(* IEC 61131-3 sources: SmartHomeNew/ (part 8) *)

(* ---- FB_Rule_Engine.st ---- *)
FUNCTION_BLOCK FB_Rule_Engine
VAR_INPUT
    VI_System_Time_MS : UDINT;
    VI_IsActivePLC : BOOL;
    VI_Security_Armed : BOOL;
    VI_Current_Time : TOD;
    VI_Day_Of_Week : INT;
END_VAR
VAR_IN_OUT
    VI_Rules : ARRAY[1..GVL_CONSTANTS.C_MAX_RULES] OF ST_User_Rule;
    VI_Indoor_Temps : ARRAY[1..16] OF REAL;
    VI_Floor_Temps : ARRAY[1..GVL_CONSTANTS.C_MAX_HEATING_CIRCUITS] OF REAL;
    VI_Humidities : ARRAY[1..16] OF REAL;
    VI_CO2_Levels : ARRAY[1..16] OF REAL;
    VI_Motion_Sensors : ARRAY[1..16] OF BOOL;
    VI_Door_Sensors : ARRAY[1..GVL_CONSTANTS.C_MAX_DOOR_SENSORS] OF BOOL;
    VI_Window_Sensors : ARRAY[1..16] OF BOOL;
    VI_Water_Sensors : ARRAY[1..GVL_CONSTANTS.C_MAX_FLOOD_SENSORS] OF BOOL;
    VI_Smoke_Sensors : ARRAY[1..GVL_CONSTANTS.C_MAX_SMOKE_SENSORS] OF BOOL;
    VI_Methane_Sensors : ARRAY[1..GVL_CONSTANTS.C_MAX_METHANE_SENSORS] OF REAL;
    VI_CO_Sensors : ARRAY[1..GVL_CONSTANTS.C_MAX_CO_SENSORS] OF REAL;
END_VAR
VAR_OUTPUT
    VO_Preheat_Request : BOOL;
    VO_Actions : ARRAY[1..GVL_CONSTANTS.C_MAX_RULES] OF ST_Rule_Action;
END_VAR
VAR
    L_i : INT;
    L_Condition_Met : BOOL;
    L_Current_Value : REAL;
    L_Triggers : ARRAY[1..GVL_CONSTANTS.C_MAX_RULES] OF R_TRIG;
    L_Trigger_Count : ARRAY[1..GVL_CONSTANTS.C_MAX_RULES] OF UINT;
    L_Last_Reset_Time : UDINT;
    L_Elapsed_Time : UDINT;
END_VAR

IF NOT VI_IsActivePLC THEN
    FOR L_i := 1 TO GVL_CONSTANTS.C_MAX_RULES DO
        VO_Actions[L_i].Active := FALSE;
        VO_Actions[L_i].Triggered := FALSE;
        VO_Actions[L_i].Action_Type := E_Rule_Action_Type.ACTION_NONE;
        VO_Actions[L_i].Target_ID := 0;
        VO_Actions[L_i].Value := 0.0;
    END_FOR;
    VO_Preheat_Request := FALSE;
    RETURN;
END_IF;

VO_Preheat_Request := FALSE;

L_Elapsed_Time := SEL(VI_System_Time_MS >= L_Last_Reset_Time, VI_System_Time_MS - L_Last_Reset_Time, (4294967295 - L_Last_Reset_Time) + VI_System_Time_MS + 1);

IF L_Elapsed_Time >= GVL_CONSTANTS.C_MS_IN_MINUTE THEN
    L_Last_Reset_Time := VI_System_Time_MS;
    FOR L_i := 1 TO GVL_CONSTANTS.C_MAX_RULES DO
        L_Trigger_Count[L_i] := 0;
    END_FOR;
END_IF;

FOR L_i := 1 TO GVL_CONSTANTS.C_MAX_RULES DO

    // Full per-cycle action reset prevents stale Triggered/Action_Type/Target_ID/Value
    // from being observed by any downstream consumer when a rule is disabled or inactive.
    VO_Actions[L_i].Active := FALSE;
    VO_Actions[L_i].Triggered := FALSE;
    VO_Actions[L_i].Action_Type := E_Rule_Action_Type.ACTION_NONE;
    VO_Actions[L_i].Target_ID := 0;
    VO_Actions[L_i].Value := 0.0;

    IF VI_Rules[L_i].Enabled THEN
        L_Condition_Met := FALSE;
        L_Current_Value := 0.0;

        IF VI_Rules[L_i].Condition_Target_ID > 0 THEN
            CASE VI_Rules[L_i].Condition_Type OF
                E_Rule_Condition_Type.COND_AIR_TEMP:
                    IF VI_Rules[L_i].Condition_Target_ID <= 16 THEN
                        L_Current_Value := VI_Indoor_Temps[VI_Rules[L_i].Condition_Target_ID];
                    END_IF;
                E_Rule_Condition_Type.COND_FLOOR_TEMP:
                    IF VI_Rules[L_i].Condition_Target_ID <= GVL_CONSTANTS.C_MAX_HEATING_CIRCUITS THEN
                        L_Current_Value := VI_Floor_Temps[VI_Rules[L_i].Condition_Target_ID];
                    END_IF;
                E_Rule_Condition_Type.COND_HUMIDITY:
                    IF VI_Rules[L_i].Condition_Target_ID <= 16 THEN
                        L_Current_Value := VI_Humidities[VI_Rules[L_i].Condition_Target_ID];
                    END_IF;
                E_Rule_Condition_Type.COND_CO2:
                    IF VI_Rules[L_i].Condition_Target_ID <= 16 THEN
                        L_Current_Value := VI_CO2_Levels[VI_Rules[L_i].Condition_Target_ID];
                    END_IF;
                E_Rule_Condition_Type.COND_MOTION:
                    IF VI_Rules[L_i].Condition_Target_ID <= 16 THEN
                        L_Current_Value := SEL(VI_Motion_Sensors[VI_Rules[L_i].Condition_Target_ID], 0.0, 1.0);
                    END_IF;
                E_Rule_Condition_Type.COND_DOOR_WINDOW:
                    IF VI_Rules[L_i].Condition_Target_ID <= GVL_CONSTANTS.C_MAX_DOOR_SENSORS THEN
                        L_Current_Value := SEL(VI_Door_Sensors[VI_Rules[L_i].Condition_Target_ID] OR VI_Window_Sensors[VI_Rules[L_i].Condition_Target_ID], 0.0, 1.0);
                    ELSIF VI_Rules[L_i].Condition_Target_ID <= 16 THEN
                        L_Current_Value := SEL(VI_Window_Sensors[VI_Rules[L_i].Condition_Target_ID], 0.0, 1.0);
                    END_IF;
                E_Rule_Condition_Type.COND_FLOOD:
                    IF VI_Rules[L_i].Condition_Target_ID <= GVL_CONSTANTS.C_MAX_FLOOD_SENSORS THEN
                        L_Current_Value := SEL(VI_Water_Sensors[VI_Rules[L_i].Condition_Target_ID], 0.0, 1.0);
                    END_IF;
                E_Rule_Condition_Type.COND_SMOKE:
                    IF VI_Rules[L_i].Condition_Target_ID <= GVL_CONSTANTS.C_MAX_SMOKE_SENSORS THEN
                        L_Current_Value := SEL(VI_Smoke_Sensors[VI_Rules[L_i].Condition_Target_ID], 0.0, 1.0);
                    END_IF;
                E_Rule_Condition_Type.COND_METHANE:
                    IF VI_Rules[L_i].Condition_Target_ID <= GVL_CONSTANTS.C_MAX_METHANE_SENSORS THEN
                        L_Current_Value := VI_Methane_Sensors[VI_Rules[L_i].Condition_Target_ID];
                    END_IF;
                E_Rule_Condition_Type.COND_CO:
                    IF VI_Rules[L_i].Condition_Target_ID <= GVL_CONSTANTS.C_MAX_CO_SENSORS THEN
                        L_Current_Value := VI_CO_Sensors[VI_Rules[L_i].Condition_Target_ID];
                    END_IF;
                E_Rule_Condition_Type.COND_TIME_OF_DAY:
                    L_Current_Value := TO_REAL(TOD_TO_UDINT(VI_Current_Time) / GVL_CONSTANTS.C_MS_IN_MINUTE);
                E_Rule_Condition_Type.COND_DAY_OF_WEEK:
                    L_Current_Value := TO_REAL(VI_Day_Of_Week);
            END_CASE;
        ELSE
            IF VI_Rules[L_i].Condition_Type = E_Rule_Condition_Type.COND_TIME_OF_DAY THEN
                L_Current_Value := TO_REAL(TOD_TO_UDINT(VI_Current_Time) / GVL_CONSTANTS.C_MS_IN_MINUTE);
            ELSIF VI_Rules[L_i].Condition_Type = E_Rule_Condition_Type.COND_DAY_OF_WEEK THEN
                L_Current_Value := TO_REAL(VI_Day_Of_Week);
            END_IF;
        END_IF;

        CASE VI_Rules[L_i].Condition_Op OF
            E_Rule_Comparison.COMP_GT:
                L_Condition_Met := (L_Current_Value > VI_Rules[L_i].Condition_Value);
            E_Rule_Comparison.COMP_LT:
                L_Condition_Met := (L_Current_Value < VI_Rules[L_i].Condition_Value);
            E_Rule_Comparison.COMP_EQ:
                L_Condition_Met := (ABS(L_Current_Value - VI_Rules[L_i].Condition_Value) < 0.1);
            E_Rule_Comparison.COMP_GE:
                L_Condition_Met := (L_Current_Value >= VI_Rules[L_i].Condition_Value);
            E_Rule_Comparison.COMP_LE:
                L_Condition_Met := (L_Current_Value <= VI_Rules[L_i].Condition_Value);
            E_Rule_Comparison.COMP_IN_RANGE:
                L_Condition_Met := (L_Current_Value >= VI_Rules[L_i].Condition_Value) AND (L_Current_Value <= VI_Rules[L_i].Condition_Value_Max);
            E_Rule_Comparison.COMP_TRUE:
                L_Condition_Met := (L_Current_Value > 0.5);
            E_Rule_Comparison.COMP_FALSE:
                L_Condition_Met := (L_Current_Value < 0.5);
        END_CASE;

        L_Triggers[L_i](CLK := L_Condition_Met);

        IF L_Triggers[L_i].Q THEN
            L_Trigger_Count[L_i] := L_Trigger_Count[L_i] + 1;
            IF L_Trigger_Count[L_i] > 10 THEN
                CONTINUE;
            END_IF;
        END_IF;

        IF L_Condition_Met AND (L_Trigger_Count[L_i] <= 10) THEN
            VO_Actions[L_i].Active := TRUE;
            VO_Actions[L_i].Triggered := L_Triggers[L_i].Q;
            VO_Actions[L_i].Action_Type := VI_Rules[L_i].Action_Type;
            VO_Actions[L_i].Target_ID := VI_Rules[L_i].Action_Target_ID;
            VO_Actions[L_i].Value := VI_Rules[L_i].Action_Value;

            // Bridge rule-driven heating intent to policy. Per-circuit valve
            // projection remains owned by FB_Heating_Circuit_Control.
            IF (VI_Rules[L_i].Action_Type = E_Rule_Action_Type.ACTION_SET_FLOOR_HEATING) AND
               (VI_Rules[L_i].Action_Value > REAL#0.5) THEN
                VO_Preheat_Request := TRUE;
            END_IF;
        END_IF;
    END_IF;
END_FOR;

// >>> BULK_SYNC_ANCHOR: FB_Rule_Engine <<<
END_FUNCTION_BLOCK

(* ---- FB_Runtime_Bus_Replication.st ---- *)
FUNCTION_BLOCK FB_Runtime_Bus_Replication
VAR_INPUT
    VI_Enable : BOOL;
    VI_System_Time_MS : UDINT;
END_VAR
VAR
    L_Frame : ST_Runtime_Bus_Frame;
    L_TX_Index : UINT;

    L_Finalized_Runtime_Continuity : BOOL;
END_VAR

IF NOT VI_Enable THEN
    GVL_Runtime_Bus.G_Runtime_Valid := FALSE;
    RETURN;
END_IF;

// Finalized runtime continuity proof chain.
L_Finalized_Runtime_Continuity :=
    GVL_SEMANTIC_PROGRESS.Semantic_Forward_Progress_Valid
    AND GVL_SEMANTIC_PROGRESS.Semantic_Execution_Continuity_OK
    AND NOT GVL_SEMANTIC_PROGRESS.Semantic_Progress_Lease_Expired
    AND NOT GVL_SEMANTIC_PROGRESS.Semantic_Progress_Quarantine_Active
    AND GVL_RUNTIME_SNAPSHOT.Snapshot_Frozen
    AND GVL_RUNTIME_SNAPSHOT.Snapshot_Publication_Allowed
    AND GVL_RUNTIME_SNAPSHOT.Snapshot_Copy_Valid
    AND GVL_RUNTIME_SNAPSHOT.Snapshot_Isolation_Valid
    AND NOT GVL_RUNTIME_SNAPSHOT.Snapshot_Mutation_Detected
    AND GVL_DISTRIBUTED_SNAPSHOT.Distributed_Publication_Reconciled
    AND GVL_DISTRIBUTED_SNAPSHOT.Distributed_Publication_Freeze_Valid
    AND GVL_DISTRIBUTED_SNAPSHOT.Distributed_Snapshot_Consistent
    AND GVL_DISTRIBUTED_COMMIT.Distributed_Commit_Valid
    AND GVL_DISTRIBUTED_COMMIT.Publication_Prepare_Valid
    AND GVL_DISTRIBUTED_COMMIT.Publication_Commit_Confirmed
    AND NOT GVL_DISTRIBUTED_COMMIT.Peer_Commit_Mismatch
    AND NOT GVL_DISTRIBUTED_COMMIT.Commit_Lease_Expired
    AND GVL_OUTPUT_EPOCH.Output_Publication_Valid
    AND GVL_OUTPUT_EPOCH.Output_Runtime_Epoch_Valid
    AND NOT GVL_OUTPUT_EPOCH.Output_Lease_Expired
    AND NOT GVL_OUTPUT_EPOCH.Output_Forced_Safe_Decay
    AND GVL_COMMAND_VERIFY.PreOutput_Barrier_OK
    AND NOT GVL_COMMAND_VERIFY.PreOutput_Block_IO;

// Deterministic runtime replication frame publication.
L_TX_Index := GVL_Runtime_Bus.G_Last_Sequence_Id + 1;

IF L_TX_Index > 128 THEN
    L_TX_Index := 1;
END_IF;

L_Frame := (Frame_Valid := TRUE);

L_Frame.Frame_Time_MS := VI_System_Time_MS;
L_Frame.Frame_Id := GVL_Runtime_Bus.G_Last_Frame_Id + 1;

L_Frame.Source_Controller_Id :=
    GVL_Distributed_Runtime.G_Local_Node_State.Controller_Id;

L_Frame.Source_Runtime_Node_Id :=
    GVL_Distributed_Runtime.G_Local_Node_State.Runtime_Node_Id;

L_Frame.Frame_Sequence_Id :=
    GVL_Runtime_Bus.G_Last_Sequence_Id + 1;

L_Frame.Frame_Ack_Required := TRUE;

// Replicated semantic domains.
L_Frame.Authority_State_Frame := TRUE;
L_Frame.Recovery_State_Frame := TRUE;
L_Frame.Quarantine_State_Frame := TRUE;
L_Frame.Topology_State_Frame := TRUE;
L_Frame.Binding_State_Frame := TRUE;
L_Frame.Predictive_State_Frame := TRUE;

// Deterministic replication safety.
IF GVL_Distributed_Authority.G_Distributed_Safety_Barrier_OK
   AND NOT GVL_Distributed_Runtime.G_Split_Brain_Suspected
   AND L_Finalized_Runtime_Continuity THEN

    L_Frame.Replication_Consistent := TRUE;

    L_Frame.Status_Code := 0;
    L_Frame.Status_Text :=
        'Deterministic replication frame accepted';

ELSE

    L_Frame.Replication_Rejected := TRUE;

    L_Frame.Status_Code := 2;
    L_Frame.Status_Text :=
        'Deterministic replication frame rejected';

END_IF;

GVL_Runtime_Bus.G_TX_Frames[L_TX_Index] := L_Frame;

GVL_Runtime_Bus.G_Last_Frame_Id :=
    L_Frame.Frame_Id;

GVL_Runtime_Bus.G_Last_Sequence_Id :=
    L_Frame.Frame_Sequence_Id;

GVL_Runtime_Bus.G_TX_Healthy :=
    L_Frame.Replication_Consistent;

GVL_Runtime_Bus.G_RX_Healthy := TRUE;

GVL_Runtime_Bus.G_Any_Replication_Rejected :=
    L_Frame.Replication_Rejected;

GVL_Runtime_Bus.G_Runtime_Valid := TRUE;
GVL_Runtime_Bus.G_Last_Update_MS := VI_System_Time_MS;

IF L_Frame.Replication_Rejected THEN
    GVL_Runtime_Bus.G_Status_Code := 2;
    GVL_Runtime_Bus.G_Status_Text :=
        'Runtime bus replication rejected';
ELSE
    GVL_Runtime_Bus.G_Status_Code := 0;
    GVL_Runtime_Bus.G_Status_Text :=
        'Runtime bus replication healthy';
END_IF;

END_FUNCTION_BLOCK

(* ---- FB_Runtime_Node_Discovery.st ---- *)
FUNCTION_BLOCK FB_Runtime_Node_Discovery
VAR_INPUT
    VI_Enable : BOOL;
    VI_System_Time_MS : UDINT;
END_VAR
VAR
    L_i : INT;
    L_State : ST_Runtime_Node_Discovery_State;

    L_Any_Quarantine : BOOL;
    L_Any_Rejected : BOOL;
END_VAR

IF NOT VI_Enable THEN
    GVL_Runtime_Discovery.G_Runtime_Valid := FALSE;
    RETURN;
END_IF;

FOR L_i := 1 TO 32 DO

    L_State := GVL_Runtime_Discovery.G_Discovery_State[L_i];

    IF L_State.Discovery_Active THEN

        L_State.Runtime_Valid := TRUE;
        L_State.Runtime_System_Time_MS := VI_System_Time_MS;

        L_State.Node_Discovered := TRUE;

        IF GVL_Distributed_Authority.G_Distributed_Safety_Barrier_OK
           AND NOT GVL_Runtime_Sessions.G_Any_Stale_Session THEN

            L_State.Node_Validated := TRUE;
            L_State.Node_Authorized := TRUE;

            L_State.Capability_Validated := TRUE;
            L_State.Execution_Domain_Assigned := TRUE;
            L_State.Deployment_Assigned := TRUE;

            L_State.Status_Code := 0;
            L_State.Status_Text :=
                'Runtime node discovery healthy';

        ELSE

            L_State.Node_Quarantined := TRUE;
            L_State.Discovery_Rejected := TRUE;

            L_Any_Quarantine := TRUE;
            L_Any_Rejected := TRUE;

            L_State.Status_Code := 2;
            L_State.Status_Text :=
                'Runtime node discovery rejected';

        END_IF;

        GVL_Runtime_Discovery.G_Discovery_State[L_i] :=
            L_State;

    END_IF;

END_FOR;

GVL_Runtime_Discovery.G_Any_Node_Quarantined :=
    L_Any_Quarantine;

GVL_Runtime_Discovery.G_Any_Discovery_Rejected :=
    L_Any_Rejected;

GVL_Runtime_Discovery.G_Runtime_Valid := TRUE;
GVL_Runtime_Discovery.G_Last_Update_MS := VI_System_Time_MS;

IF L_Any_Rejected THEN
    GVL_Runtime_Discovery.G_Status_Code := 2;
    GVL_Runtime_Discovery.G_Status_Text :=
        'Runtime discovery rejection detected';
ELSIF L_Any_Quarantine THEN
    GVL_Runtime_Discovery.G_Status_Code := 1;
    GVL_Runtime_Discovery.G_Status_Text :=
        'Runtime discovery quarantine active';
ELSE
    GVL_Runtime_Discovery.G_Status_Code := 0;
    GVL_Runtime_Discovery.G_Status_Text :=
        'Runtime discovery governance healthy';
END_IF;

END_FUNCTION_BLOCK

(* ---- FB_Runtime_Restart_Continuity.st ---- *)
FUNCTION_BLOCK FB_Runtime_Restart_Continuity
VAR_INPUT
    VI_Enable : BOOL;
    VI_System_Time_MS : UDINT;
    VI_Warm_Restart : BOOL;
END_VAR
VAR
    L_State : ST_Runtime_Restart_Continuity_State;
END_VAR

IF NOT VI_Enable THEN
    GVL_Runtime_Restart_Continuity.G_Runtime_Valid := FALSE;
    RETURN;
END_IF;

L_State := (Runtime_Valid := TRUE);
L_State.Runtime_System_Time_MS := VI_System_Time_MS;

L_State.Warm_Restart_Detected := VI_Warm_Restart;
L_State.Cold_Start_Detected := NOT VI_Warm_Restart;

L_State.Active_Config_Version :=
    GVL_Water_Topology_Config.G_Active_Config_Version;

L_State.Restored_Config_Version :=
    GVL_Runtime_Restart_Continuity.G_Last_Stable_Config_Version;

L_State.Last_Stable_Config_Version :=
    GVL_Runtime_Restart_Continuity.G_Last_Stable_Config_Version;

L_State.Restore_Requested :=
    GVL_Runtime_Restart_Continuity.G_Restore_Request;

L_State.Post_Restart_Validation_Required :=
    GVL_Runtime_Restart_Continuity.G_Post_Restart_Validation_Request;

L_State.Retained_State_Valid := TRUE;
L_State.Topology_Restore_Valid := TRUE;
L_State.Config_Restore_Valid := TRUE;
L_State.Recovery_Restore_Valid := TRUE;
L_State.Quarantine_Restore_Valid := TRUE;

IF L_State.Restore_Requested THEN

    IF L_State.Retained_State_Valid
       AND L_State.Topology_Restore_Valid
       AND L_State.Config_Restore_Valid THEN

        L_State.Restore_Allowed := TRUE;
        L_State.Restore_Completed := TRUE;

        GVL_Config_Activation.G_Config_Quarantine_Active :=
            GVL_Runtime_Restart_Continuity.G_Last_Known_Quarantine_State;

        L_State.Status_Code := 1;
        L_State.Status_Text := 'Runtime continuity restored';

    ELSE

        L_State.Restore_Blocked := TRUE;
        L_State.Safe_Mode_Required := TRUE;
        L_State.Operator_Ack_Required := TRUE;

        L_State.Status_Code := 2;
        L_State.Status_Text := 'Runtime continuity restore blocked';

    END_IF;

ELSIF L_State.Post_Restart_Validation_Required THEN

    IF GVL_Water_Runtime_Hardening.G_Runtime_Valid
       AND GVL_Water_Output_Reconciliation.G_Runtime_Valid
       AND NOT GVL_Water_Output_Reconciliation.G_Any_Conflict_Detected THEN

        L_State.Post_Restart_Validation_OK := TRUE;

        L_State.Status_Code := 0;
        L_State.Status_Text := 'Post-restart validation healthy';

    ELSE

        L_State.Post_Restart_Validation_Failed := TRUE;
        L_State.Safe_Mode_Required := TRUE;

        L_State.Status_Code := 3;
        L_State.Status_Text := 'Post-restart validation failed';

    END_IF;

ELSE

    L_State.Status_Code := 0;
    L_State.Status_Text := 'Runtime restart continuity healthy';

END_IF;

GVL_Runtime_Restart_Continuity.G_Continuity_State := L_State;

GVL_Runtime_Restart_Continuity.G_Runtime_Valid := TRUE;
GVL_Runtime_Restart_Continuity.G_Last_Update_MS := VI_System_Time_MS;
GVL_Runtime_Restart_Continuity.G_Status_Code := L_State.Status_Code;
GVL_Runtime_Restart_Continuity.G_Status_Text := L_State.Status_Text;

END_FUNCTION_BLOCK

(* ---- FB_Runtime_Session_Governance.st ---- *)
FUNCTION_BLOCK FB_Runtime_Session_Governance
VAR_INPUT
    VI_Enable : BOOL;
    VI_System_Time_MS : UDINT;
END_VAR
VAR
    L_i : INT;
    L_Session : ST_Runtime_Node_Session;
    L_Any_Stale : BOOL;
    L_Any_Quarantine : BOOL;

    L_Finalized_Runtime_Continuity : BOOL;
END_VAR

IF NOT VI_Enable THEN
    GVL_Runtime_Sessions.G_Runtime_Valid := FALSE;
    RETURN;
END_IF;

// Finalized runtime continuity proof chain.
L_Finalized_Runtime_Continuity :=
    GVL_SEMANTIC_PROGRESS.Semantic_Forward_Progress_Valid
    AND GVL_SEMANTIC_PROGRESS.Semantic_Execution_Continuity_OK
    AND NOT GVL_SEMANTIC_PROGRESS.Semantic_Progress_Lease_Expired
    AND NOT GVL_SEMANTIC_PROGRESS.Semantic_Progress_Quarantine_Active
    AND GVL_RUNTIME_SNAPSHOT.Snapshot_Frozen
    AND GVL_RUNTIME_SNAPSHOT.Snapshot_Publication_Allowed
    AND GVL_RUNTIME_SNAPSHOT.Snapshot_Copy_Valid
    AND GVL_RUNTIME_SNAPSHOT.Snapshot_Isolation_Valid
    AND NOT GVL_RUNTIME_SNAPSHOT.Snapshot_Mutation_Detected
    AND GVL_DISTRIBUTED_SNAPSHOT.Distributed_Publication_Reconciled
    AND GVL_DISTRIBUTED_SNAPSHOT.Distributed_Publication_Freeze_Valid
    AND GVL_DISTRIBUTED_SNAPSHOT.Distributed_Snapshot_Consistent
    AND GVL_DISTRIBUTED_COMMIT.Distributed_Commit_Valid
    AND GVL_DISTRIBUTED_COMMIT.Publication_Prepare_Valid
    AND GVL_DISTRIBUTED_COMMIT.Publication_Commit_Confirmed
    AND NOT GVL_DISTRIBUTED_COMMIT.Peer_Commit_Mismatch
    AND NOT GVL_DISTRIBUTED_COMMIT.Commit_Lease_Expired
    AND GVL_OUTPUT_EPOCH.Output_Publication_Valid
    AND GVL_OUTPUT_EPOCH.Output_Runtime_Epoch_Valid
    AND NOT GVL_OUTPUT_EPOCH.Output_Lease_Expired
    AND NOT GVL_OUTPUT_EPOCH.Output_Forced_Safe_Decay
    AND GVL_COMMAND_VERIFY.PreOutput_Barrier_OK
    AND NOT GVL_COMMAND_VERIFY.PreOutput_Block_IO;

GVL_Runtime_Sessions.G_Local_Session.Session_Valid := TRUE;
GVL_Runtime_Sessions.G_Local_Session.Session_Connected := TRUE;
GVL_Runtime_Sessions.G_Local_Session.Last_Heartbeat_MS :=
    VI_System_Time_MS;

GVL_Runtime_Sessions.G_Local_Session.Transport_Healthy :=
    GVL_Runtime_Bus.G_TX_Healthy
    AND L_Finalized_Runtime_Continuity;

GVL_Runtime_Sessions.G_Local_Session.Runtime_Replication_Healthy :=
    GVL_Distributed_Runtime.G_Distributed_Replication_Healthy
    AND L_Finalized_Runtime_Continuity;

GVL_Runtime_Sessions.G_Local_Session.Authority_Granted :=
    GVL_Distributed_Authority.G_Authority_State.Authority_Master_Elected
    AND L_Finalized_Runtime_Continuity;

FOR L_i := 1 TO 16 DO

    L_Session := GVL_Runtime_Sessions.G_Remote_Sessions[L_i];

    IF L_Session.Session_Valid THEN

        IF (VI_System_Time_MS - L_Session.Last_Heartbeat_MS) > 30000 THEN

            L_Session.Session_Stale := TRUE;
            L_Session.Session_Reconnect_Required := TRUE;

            L_Any_Stale := TRUE;

        END_IF;

        IF NOT L_Finalized_Runtime_Continuity THEN

            L_Session.Session_Stale := TRUE;
            L_Session.Session_Quarantined := TRUE;

            L_Any_Stale := TRUE;
            L_Any_Quarantine := TRUE;

        END_IF;

        IF L_Session.Session_Quarantined THEN
            L_Any_Quarantine := TRUE;
        END_IF;

        GVL_Runtime_Sessions.G_Remote_Sessions[L_i] :=
            L_Session;

    END_IF;

END_FOR;

GVL_Runtime_Sessions.G_Any_Stale_Session :=
    L_Any_Stale;

GVL_Runtime_Sessions.G_Any_Quarantined_Session :=
    L_Any_Quarantine;

GVL_Runtime_Sessions.G_Runtime_Valid := TRUE;
GVL_Runtime_Sessions.G_Last_Update_MS := VI_System_Time_MS;

IF L_Any_Quarantine THEN
    GVL_Runtime_Sessions.G_Status_Code := 2;
    GVL_Runtime_Sessions.G_Status_Text :=
        'Quarantined runtime session detected';
ELSIF L_Any_Stale THEN
    GVL_Runtime_Sessions.G_Status_Code := 1;
    GVL_Runtime_Sessions.G_Status_Text :=
        'Stale runtime session detected';
ELSE
    GVL_Runtime_Sessions.G_Status_Code := 0;
    GVL_Runtime_Sessions.G_Status_Text :=
        'Runtime session governance healthy';
END_IF;

END_FUNCTION_BLOCK

(* ---- FB_Safety_Workflow_Manager.st ---- *)
FUNCTION_BLOCK FB_Safety_Workflow_Manager
VAR_INPUT
    VI_System_Time_MS : UDINT;
    VI_Water_Selective_Recover : BOOL;
    VI_Gas_Selective_Recover : BOOL;
    VI_Water_Valve_Test_Open : BOOL;
    VI_Water_Valve_Test_Close : BOOL;
    VI_Water_Valve_Test_Confirm : BOOL;
    VI_Gas_Valve_Test_Open : BOOL;
    VI_Gas_Valve_Test_Close : BOOL;
    VI_Gas_Valve_Test_Confirm : BOOL;
END_VAR
VAR_OUTPUT
    VO_Water_Selective_Recover_Edge : BOOL;
    VO_Gas_Selective_Recover_Edge : BOOL;
    VO_Water_Valve_Test_Open_Edge : BOOL;
    VO_Water_Valve_Test_Close_Edge : BOOL;
    VO_Water_Valve_Test_Confirm_Edge : BOOL;
    VO_Gas_Valve_Test_Open_Edge : BOOL;
    VO_Gas_Valve_Test_Close_Edge : BOOL;
    VO_Gas_Valve_Test_Confirm_Edge : BOOL;
    VO_Water_Test_Active : BOOL;
    VO_Gas_Test_Active : BOOL;
    VO_Water_Test_Timeout_Close_Required : BOOL;
    VO_Gas_Test_Timeout_Close_Required : BOOL;
END_VAR
VAR
    L_CMD_Water_Selective_Recover_Prev : BOOL;
    L_CMD_Gas_Selective_Recover_Prev : BOOL;
    L_CMD_Water_Valve_Test_Open_Prev : BOOL;
    L_CMD_Water_Valve_Test_Close_Prev : BOOL;
    L_CMD_Water_Valve_Test_Confirm_Prev : BOOL;
    L_CMD_Gas_Valve_Test_Open_Prev : BOOL;
    L_CMD_Gas_Valve_Test_Close_Prev : BOOL;
    L_CMD_Gas_Valve_Test_Confirm_Prev : BOOL;
    L_Water_Test_Active : BOOL;
    L_Water_Test_Start_MS : UDINT;
    L_Gas_Test_Active : BOOL;
    L_Gas_Test_Start_MS : UDINT;
END_VAR

VO_Water_Test_Timeout_Close_Required := FALSE;
VO_Gas_Test_Timeout_Close_Required := FALSE;

VO_Water_Selective_Recover_Edge := VI_Water_Selective_Recover AND NOT L_CMD_Water_Selective_Recover_Prev;
VO_Gas_Selective_Recover_Edge := VI_Gas_Selective_Recover AND NOT L_CMD_Gas_Selective_Recover_Prev;
VO_Water_Valve_Test_Open_Edge := VI_Water_Valve_Test_Open AND NOT L_CMD_Water_Valve_Test_Open_Prev;
VO_Water_Valve_Test_Close_Edge := VI_Water_Valve_Test_Close AND NOT L_CMD_Water_Valve_Test_Close_Prev;
VO_Water_Valve_Test_Confirm_Edge := VI_Water_Valve_Test_Confirm AND NOT L_CMD_Water_Valve_Test_Confirm_Prev;
VO_Gas_Valve_Test_Open_Edge := VI_Gas_Valve_Test_Open AND NOT L_CMD_Gas_Valve_Test_Open_Prev;
VO_Gas_Valve_Test_Close_Edge := VI_Gas_Valve_Test_Close AND NOT L_CMD_Gas_Valve_Test_Close_Prev;
VO_Gas_Valve_Test_Confirm_Edge := VI_Gas_Valve_Test_Confirm AND NOT L_CMD_Gas_Valve_Test_Confirm_Prev;

L_CMD_Water_Selective_Recover_Prev := VI_Water_Selective_Recover;
L_CMD_Gas_Selective_Recover_Prev := VI_Gas_Selective_Recover;
L_CMD_Water_Valve_Test_Open_Prev := VI_Water_Valve_Test_Open;
L_CMD_Water_Valve_Test_Close_Prev := VI_Water_Valve_Test_Close;
L_CMD_Water_Valve_Test_Confirm_Prev := VI_Water_Valve_Test_Confirm;
L_CMD_Gas_Valve_Test_Open_Prev := VI_Gas_Valve_Test_Open;
L_CMD_Gas_Valve_Test_Close_Prev := VI_Gas_Valve_Test_Close;
L_CMD_Gas_Valve_Test_Confirm_Prev := VI_Gas_Valve_Test_Confirm;

IF VO_Water_Valve_Test_Open_Edge THEN
    L_Water_Test_Active := TRUE;
    L_Water_Test_Start_MS := VI_System_Time_MS;
END_IF;

IF VO_Water_Valve_Test_Close_Edge OR VO_Water_Valve_Test_Confirm_Edge THEN
    L_Water_Test_Active := FALSE;
END_IF;

IF L_Water_Test_Active THEN
    IF (VI_System_Time_MS - L_Water_Test_Start_MS) >= 60000 THEN
        L_Water_Test_Active := FALSE;
        VO_Water_Test_Timeout_Close_Required := TRUE;
    END_IF;
END_IF;

IF VO_Gas_Valve_Test_Open_Edge THEN
    L_Gas_Test_Active := TRUE;
    L_Gas_Test_Start_MS := VI_System_Time_MS;
END_IF;

IF VO_Gas_Valve_Test_Close_Edge OR VO_Gas_Valve_Test_Confirm_Edge THEN
    L_Gas_Test_Active := FALSE;
END_IF;

IF L_Gas_Test_Active THEN
    IF (VI_System_Time_MS - L_Gas_Test_Start_MS) >= 60000 THEN
        L_Gas_Test_Active := FALSE;
        VO_Gas_Test_Timeout_Close_Required := TRUE;
    END_IF;
END_IF;

VO_Water_Test_Active := L_Water_Test_Active;
VO_Gas_Test_Active := L_Gas_Test_Active;
END_FUNCTION_BLOCK

(* ---- FB_Scenario_Manager.st ---- *)
FUNCTION_BLOCK FB_Scenario_Manager
VAR_INPUT
    VI_Preheat_Request : BOOL;
    VI_System_Time_MS : UDINT; // Системное время (мс)
    VI_Activate_Request : E_SCENARIO_TYPE; // Запрос на активацию сценария
    VI_IsActivePLC : BOOL; // Флаг: Данный ПЛК является ведущим
    VI_System_Mode : E_System_Operating_Mode; // Агрегированный режим работы системы
END_VAR
VAR_OUTPUT
    VO_Current_Scenario : E_SCENARIO_TYPE; // Текущий активный сценарий
    VO_Status_Msg : STRING(200); // Строковое сообщение о статусе
END_VAR

VAR
    L_Last_Scenario_Time : UDINT;
END_VAR

IF NOT VI_IsActivePLC THEN
    RETURN;
END_IF;

CASE VI_System_Mode OF
    E_System_Operating_Mode.MODE_SAFE_STOP,
    E_System_Operating_Mode.MODE_FREEZE_PROTECTION:
        IF VO_Current_Scenario <> E_SCENARIO_TYPE.SCENARIO_NONE THEN
            VO_Current_Scenario := E_SCENARIO_TYPE.SCENARIO_NONE;
            VO_Status_Msg := 'Сценарии принудительно отключены режимом безопасности';
        END_IF;
        RETURN;

    E_System_Operating_Mode.MODE_DEGRADED:
        VO_Status_Msg := 'Смена сценариев заблокирована: деградированный режим';
        RETURN;
ELSE
        // No fallback required
END_CASE;

IF VI_Activate_Request <> VO_Current_Scenario THEN
    // Проверка минимального времени работы сценария
    IF (VI_System_Time_MS - L_Last_Scenario_Time) >= 60000 OR VO_Current_Scenario = E_SCENARIO_TYPE.SCENARIO_NONE THEN
        // Логика переключения сценариев
        VO_Current_Scenario := VI_Activate_Request;
        L_Last_Scenario_Time := VI_System_Time_MS;

        CASE VO_Current_Scenario OF
        E_SCENARIO_TYPE.SCENARIO_NONE:
            VO_Status_Msg := 'Сценарии отключены';
        E_SCENARIO_TYPE.SCENARIO_AWAY:
            VO_Status_Msg := 'Активирован сценарий: Вне дома (Охрана + Энергосбережение)';
        E_SCENARIO_TYPE.SCENARIO_SLEEP:
            VO_Status_Msg := 'Активирован сценарий: Сон (Ночное освещение + Климат)';
        E_SCENARIO_TYPE.SCENARIO_PRESENCE:
            VO_Status_Msg := 'Активирован сценарий: Имитация присутствия';
        ELSE
        // No fallback required
END_CASE;
    END_IF;
END_IF;
// >>> BULK_SYNC_ANCHOR: FB_Scenario_Manager <<<

// --- PREHEAT SCENARIO INSERT ---
IF VI_Preheat_Request THEN
    // removed: direct heating write (moved to Heating Manager)
END_IF;
END_FUNCTION_BLOCK

(* ---- FB_Scenario_Transition_Guard.st ---- *)
FUNCTION_BLOCK FB_Scenario_Transition_Guard
VAR_INPUT
    VI_Current_Scenario : E_SCENARIO_TYPE;
    VI_Target_Scenario  : E_SCENARIO_TYPE;
END_VAR

VAR_OUTPUT
    VO_Transition_Allowed : BOOL;
    VO_Reason             : STRING(120);
END_VAR

VO_Transition_Allowed := TRUE;
VO_Reason := 'OK';

// no-op transition is always allowed
IF VI_Current_Scenario = VI_Target_Scenario THEN
    RETURN;
END_IF;

// emergency can always be entered
IF VI_Target_Scenario = E_SCENARIO_TYPE.SCENARIO_EMERGENCY THEN
    RETURN;
END_IF;

// from NONE, any target is allowed
IF VI_Current_Scenario = E_SCENARIO_TYPE.SCENARIO_NONE THEN
    RETURN;
END_IF;

// emergency exit is restricted
IF VI_Current_Scenario = E_SCENARIO_TYPE.SCENARIO_EMERGENCY THEN
    CASE VI_Target_Scenario OF
        E_SCENARIO_TYPE.SCENARIO_NONE,
        E_SCENARIO_TYPE.SCENARIO_AWAY,
        E_SCENARIO_TYPE.SCENARIO_SLEEP,
        E_SCENARIO_TYPE.SCENARIO_PRESENCE:
            RETURN;
    ELSE
        VO_Transition_Allowed := FALSE;
        VO_Reason := 'Переход из EMERGENCY в данный сценарий запрещён';
        RETURN;
    END_CASE;
END_IF;

// away exit is restricted to safe occupancy contexts
IF VI_Current_Scenario = E_SCENARIO_TYPE.SCENARIO_AWAY THEN
    CASE VI_Target_Scenario OF
        E_SCENARIO_TYPE.SCENARIO_NONE,
        E_SCENARIO_TYPE.SCENARIO_SLEEP,
        E_SCENARIO_TYPE.SCENARIO_PRESENCE,
        E_SCENARIO_TYPE.SCENARIO_EMERGENCY:
            RETURN;
    ELSE
        VO_Transition_Allowed := FALSE;
        VO_Reason := 'Переход из AWAY в данный сценарий запрещён';
        RETURN;
    END_CASE;
END_IF;

// default: allow
RETURN;
// >>> BULK_SYNC_ANCHOR: FB_Scenario_Transition_Guard <<<

(* ---- FB_Security_System_Manager.st ---- *)
FUNCTION_BLOCK FB_Security_System_Manager
VAR_INPUT
    VI_System_Time_MS : UDINT; // Системное время (мс)
    VI_IsActivePLC : BOOL; // Флаг: Данный ПЛК является ведущим
    VI_Arm_Request : BOOL; // Запрос на постановку под охрану
    VI_Disarm_Request : BOOL; // Запрос на снятие с охраны
    VI_PIN_Code : STRING(4); // ПИН-код для авторизации
    VI_RFID_Tag : STRING(20); // RFID/NFC метка для авторизации
    VI_2FA_Code : STRING(6); // Код двухфакторной аутентификации
    VI_Config : ST_Security_Global_Config; // Конфигурация охранной системы
    VI_Current_TOD : TOD; // Текущее время суток (от FB_Astro_Timer)
END_VAR
VAR_IN_OUT
    VI_Motion_Sensors : ARRAY[1..16] OF BOOL; // Датчики движения
    VI_Door_Sensors : ARRAY[1..GVL_CONSTANTS.C_MAX_DOOR_SENSORS] OF BOOL; // Датчики открытия дверей (герконы)
    VI_Window_Sensors : ARRAY[1..16] OF BOOL; // Датчики открытия окон (герконы)
    VI_Bypass_Motion : ARRAY[1..16] OF BOOL; // Байпас датчиков движения
    VI_Bypass_Doors : ARRAY[1..GVL_CONSTANTS.C_MAX_DOOR_SENSORS] OF BOOL; // Байпас дверей
    VI_Bypass_Windows : ARRAY[1..16] OF BOOL; // Байпас окон
END_VAR
VAR_OUTPUT
    VO_Armed : BOOL; // Статус: Система под охраной
    VO_Alarm_Active : BOOL; // Статус: Тревога активна
    VO_Siren_Active : BOOL; // Команда: Включить сирену
    VO_Status_Msg : STRING(200); // Строковое сообщение о статусе
    VO_Send_Code_Req : BOOL; // Запрос на отправку кода 2FA
    VO_Code_To_Send : STRING(6); // Сгенерированный код 2FA для отправки
END_VAR
VAR
    L_i : INT;
    L_Any_Sensor_Active : BOOL;
    L_Door_Blocking_Open : BOOL;
    L_Window_Blocking_Open : BOOL;
    L_Intrusion_Active_Count : INT;
    L_Intrusion_Event_Count : INT;
    L_Arm_Delay_Timer : FB_System_Timer;
    L_Alarm_Delay_Timer : FB_System_Timer;
    L_Arming_In_Progress : BOOL;
    L_Pin_Entry_Active : BOOL;
    L_Valid_PIN : BOOL;
    fbAccessCode : FB_AccessCode_Manager;
    fbTwoFactor : FB_TwoFactor_Auth;
    L_2FA_Required : BOOL;
    L_Disarm_Pending : BOOL;
    L_Reset_2FA : BOOL;
    L_Auto_Arm_Trigger : BOOL;
    L_Max_Attempts : BYTE;
    L_PIN_Fail_Count : BYTE;
    L_Pin_Entry_Timeout_MS : UDINT;
    L_Combined_Window_MS : UDINT;
    L_Combined_Elapsed_MS : UDINT;
    L_Combined_Window_Active : BOOL;
    L_Combined_First_Event_MS : UDINT;
    L_Combined_Event_Count : INT;
    L_Allowed_Open_Windows : ARRAY[1..16] OF BOOL;
    L_Prev_Motion_Sensors : ARRAY[1..16] OF BOOL;
    L_Prev_Door_Sensors : ARRAY[1..GVL_CONSTANTS.C_MAX_DOOR_SENSORS] OF BOOL;
    L_Prev_Window_Sensors : ARRAY[1..16] OF BOOL;
    R_Trig_Auto_Arm : R_TRIG;
    R_Trig_Arm : R_TRIG;
    R_Trig_Disarm : R_TRIG;
END_VAR

IF NOT VI_IsActivePLC THEN
    VO_Armed := FALSE;
    VO_Alarm_Active := FALSE;
    VO_Siren_Active := FALSE;
    VO_Send_Code_Req := FALSE;
    VO_Code_To_Send := '';
    VO_Status_Msg := 'Охрана: резервный ПЛК';
    L_Arming_In_Progress := FALSE;
    L_Disarm_Pending := FALSE;
    L_2FA_Required := FALSE;
    L_Reset_2FA := FALSE;
    L_Pin_Entry_Active := FALSE;
    GVL_SECURITY_WORKFLOW.G_Arming_In_Progress := FALSE;
    GVL_SECURITY_WORKFLOW.G_Pin_Entry_Active := FALSE;
    GVL_SECURITY_WORKFLOW.G_Disarm_Pending := FALSE;
    GVL_SECURITY_WORKFLOW.G_2FA_Required := FALSE;
    GVL_SECURITY_WORKFLOW.G_2FA_Send_Code_Req := FALSE;
    GVL_SECURITY_WORKFLOW.G_Combined_Window_Active := FALSE;
    GVL_SECURITY_WORKFLOW.G_Combined_Event_Count := 0;
    GVL_SECURITY_WORKFLOW.G_Intrusion_Active_Count := 0;
    GVL_SECURITY_WORKFLOW.G_Intrusion_Event_Count := 0;
    GVL_SECURITY_WORKFLOW.G_Any_Sensor_Active := FALSE;
    GVL_SECURITY_WORKFLOW.G_Status_Text := VO_Status_Msg;
    GVL_SECURITY_WORKFLOW.G_Last_Update_MS := VI_System_Time_MS;
    RETURN;
END_IF;

IF VI_Config.max_access_attempts < 1 THEN
    L_Max_Attempts := 1;
ELSE
    L_Max_Attempts := VI_Config.max_access_attempts;
END_IF;

IF VI_Config.pin_entry_timeout_seconds > 0 THEN
    L_Pin_Entry_Timeout_MS := VI_Config.pin_entry_timeout_seconds * 1000;
ELSIF VI_Config.entry_delay_seconds > 0 THEN
    L_Pin_Entry_Timeout_MS := VI_Config.entry_delay_seconds * 1000;
ELSE
    L_Pin_Entry_Timeout_MS := 45000;
END_IF;

IF VI_Config.combined_alarm_window_seconds > 0 THEN
    L_Combined_Window_MS := VI_Config.combined_alarm_window_seconds * 1000;
ELSE
    L_Combined_Window_MS := 10000;
END_IF;

R_Trig_Arm(CLK := VI_Arm_Request);
R_Trig_Disarm(CLK := VI_Disarm_Request);

// 1. Проверка PIN-кода или RFID-метки через менеджер кодов
fbAccessCode(
    VI_System_Time_MS := VI_System_Time_MS,
    VI_IsActivePLC := VI_IsActivePLC,
    VI_Code_To_Check := VI_PIN_Code,
    VI_RFID_To_Check := VI_RFID_Tag,
    VI_Access_Codes := GVL_RETAIN.G_Access_Codes,
    VI_RFID_Tags := GVL_RETAIN.G_RFID_Tags,
    VO_Code_Valid => L_Valid_PIN
);

// 2. Логика постановки на охрану (с задержкой на выход)
L_Auto_Arm_Trigger := FALSE;
IF VI_Config.auto_arm_enabled THEN
    IF VI_Current_TOD >= UDINT_TO_TOD(VI_Config.auto_arm_time_ms) THEN
        L_Auto_Arm_Trigger := TRUE;
    END_IF;
END_IF;
R_Trig_Auto_Arm(CLK := L_Auto_Arm_Trigger);

IF ((R_Trig_Arm.Q AND L_Valid_PIN) OR R_Trig_Auto_Arm.Q) AND NOT VO_Armed AND NOT L_Arming_In_Progress THEN
    L_Door_Blocking_Open := FALSE;
    L_Window_Blocking_Open := FALSE;

    FOR L_i := 1 TO GVL_CONSTANTS.C_MAX_DOOR_SENSORS DO
        IF VI_Door_Sensors[L_i] AND NOT VI_Bypass_Doors[L_i] THEN
            L_Door_Blocking_Open := TRUE;
        END_IF;
    END_FOR;

    FOR L_i := 1 TO 16 DO
        IF VI_Window_Sensors[L_i] AND NOT VI_Bypass_Windows[L_i] THEN
            L_Window_Blocking_Open := TRUE;
        END_IF;
    END_FOR;

    IF NOT L_Door_Blocking_Open AND (NOT L_Window_Blocking_Open OR VI_Config.allow_short_away_open_windows) THEN
        FOR L_i := 1 TO 16 DO
            L_Allowed_Open_Windows[L_i] :=
                VI_Config.allow_short_away_open_windows
                AND VI_Window_Sensors[L_i]
                AND NOT VI_Bypass_Windows[L_i];
        END_FOR;

        L_Arming_In_Progress := TRUE;
        L_PIN_Fail_Count := 0;
        L_Pin_Entry_Active := FALSE;
        L_Combined_Window_Active := FALSE;
        L_Combined_Event_Count := 0;
        VO_Status_Msg := 'Постановка на охрану. Покиньте помещение.';
    ELSE
        IF L_Door_Blocking_Open THEN
            VO_Status_Msg := 'Ошибка постановки: Открыты двери';
        ELSE
            VO_Status_Msg := 'Ошибка постановки: Открыты окна';
        END_IF;
    END_IF;
END_IF;

L_Arm_Delay_Timer(IN := L_Arming_In_Progress, PT := TO_TIME(VI_Config.exit_delay_seconds * 1000), VI_System_Time_MS := VI_System_Time_MS);
IF L_Arm_Delay_Timer.Q THEN
    L_Arming_In_Progress := FALSE;
    VO_Armed := TRUE;
    VO_Status_Msg := 'Система под охраной';
END_IF;

// 3. Логика снятия с охраны с PIN/RFID и 2FA
IF R_Trig_Disarm.Q AND VO_Armed THEN
    IF L_Valid_PIN THEN
        L_PIN_Fail_Count := 0;

        IF VI_Config.enable_2fa THEN
            L_Disarm_Pending := TRUE;
            L_2FA_Required := TRUE;
            VO_Status_Msg := 'Ожидание 2FA для снятия с охраны';
        ELSE
            VO_Armed := FALSE;
            VO_Alarm_Active := FALSE;
            VO_Siren_Active := FALSE;
            L_Arming_In_Progress := FALSE;
            L_Pin_Entry_Active := FALSE;
            L_Combined_Window_Active := FALSE;
            L_Combined_Event_Count := 0;
            FOR L_i := 1 TO 16 DO
                L_Allowed_Open_Windows[L_i] := FALSE;
            END_FOR;
            VO_Status_Msg := 'Система снята с охраны';
        END_IF;
    ELSE
        IF L_PIN_Fail_Count < 255 THEN
            L_PIN_Fail_Count := L_PIN_Fail_Count + 1;
        END_IF;

        IF L_PIN_Fail_Count >= L_Max_Attempts THEN
            VO_Alarm_Active := TRUE;
            VO_Siren_Active := TRUE;
            VO_Status_Msg := 'ТРЕВОГА! Превышено количество попыток PIN';
        ELSE
            VO_Status_Msg := 'Неверный PIN/RFID';
        END_IF;
    END_IF;
END_IF;

fbTwoFactor(
    VI_System_Time_MS := VI_System_Time_MS,
    VI_Start_Auth := L_2FA_Required,
    VI_Method := E_TwoFactor_Method.TF_METHOD_TOTP,
    VI_User_Code := VI_2FA_Code,
    VI_Reset_Success := L_Reset_2FA
);

VO_Send_Code_Req := fbTwoFactor.VO_Send_Code_Req;
VO_Code_To_Send := fbTwoFactor.VO_Code_To_Send;

IF L_Disarm_Pending AND fbTwoFactor.VO_State.Is_Success THEN
    VO_Armed := FALSE;
    VO_Alarm_Active := FALSE;
    VO_Siren_Active := FALSE;
    L_Arming_In_Progress := FALSE;
    L_Pin_Entry_Active := FALSE;
    L_Disarm_Pending := FALSE;
    L_2FA_Required := FALSE;
    L_Reset_2FA := TRUE;
    L_Combined_Window_Active := FALSE;
    L_Combined_Event_Count := 0;
    FOR L_i := 1 TO 16 DO
        L_Allowed_Open_Windows[L_i] := FALSE;
    END_FOR;
    VO_Status_Msg := 'Система снята с охраны';
ELSIF L_Disarm_Pending AND fbTwoFactor.VO_State.Is_Locked THEN
    L_Disarm_Pending := FALSE;
    L_2FA_Required := FALSE;
    L_Reset_2FA := FALSE;
    VO_Status_Msg := 'Ошибка 2FA: Превышено количество попыток';
ELSE
    L_Reset_2FA := FALSE;
END_IF;

// 4. Логика тревоги: задержка PIN + комбинированная авария датчиков
IF VO_Armed THEN
    FOR L_i := 1 TO 16 DO
        IF L_Allowed_Open_Windows[L_i] AND NOT VI_Window_Sensors[L_i] THEN
            L_Allowed_Open_Windows[L_i] := FALSE;
        END_IF;
    END_FOR;

    L_Any_Sensor_Active := FALSE;
    L_Intrusion_Active_Count := 0;
    L_Intrusion_Event_Count := 0;

    FOR L_i := 1 TO 16 DO
        IF VI_Motion_Sensors[L_i] AND NOT VI_Bypass_Motion[L_i] THEN
            L_Any_Sensor_Active := TRUE;
            L_Intrusion_Active_Count := L_Intrusion_Active_Count + 1;
            IF NOT L_Prev_Motion_Sensors[L_i] THEN
                L_Intrusion_Event_Count := L_Intrusion_Event_Count + 1;
            END_IF;
        END_IF;
        L_Prev_Motion_Sensors[L_i] := VI_Motion_Sensors[L_i];
    END_FOR;

    FOR L_i := 1 TO GVL_CONSTANTS.C_MAX_DOOR_SENSORS DO
        IF VI_Door_Sensors[L_i] AND NOT VI_Bypass_Doors[L_i] THEN
            L_Any_Sensor_Active := TRUE;
            L_Intrusion_Active_Count := L_Intrusion_Active_Count + 1;
            IF NOT L_Prev_Door_Sensors[L_i] THEN
                L_Intrusion_Event_Count := L_Intrusion_Event_Count + 1;
            END_IF;
        END_IF;
        L_Prev_Door_Sensors[L_i] := VI_Door_Sensors[L_i];
    END_FOR;

    FOR L_i := 1 TO 16 DO
        IF VI_Window_Sensors[L_i] AND NOT VI_Bypass_Windows[L_i] AND NOT L_Allowed_Open_Windows[L_i] THEN
            L_Any_Sensor_Active := TRUE;
            L_Intrusion_Active_Count := L_Intrusion_Active_Count + 1;
            IF NOT L_Prev_Window_Sensors[L_i] THEN
                L_Intrusion_Event_Count := L_Intrusion_Event_Count + 1;
            END_IF;
        END_IF;
        L_Prev_Window_Sensors[L_i] := VI_Window_Sensors[L_i];
    END_FOR;

    IF L_Intrusion_Event_Count > 0 THEN
        IF NOT L_Combined_Window_Active THEN
            L_Combined_Window_Active := TRUE;
            L_Combined_First_Event_MS := VI_System_Time_MS;
            L_Combined_Event_Count := L_Intrusion_Event_Count;
        ELSE
            IF VI_System_Time_MS >= L_Combined_First_Event_MS THEN
                L_Combined_Elapsed_MS := VI_System_Time_MS - L_Combined_First_Event_MS;
            ELSE
                L_Combined_Elapsed_MS := (4294967295 - L_Combined_First_Event_MS) + VI_System_Time_MS + 1;
            END_IF;

            IF L_Combined_Elapsed_MS <= L_Combined_Window_MS THEN
                L_Combined_Event_Count := L_Combined_Event_Count + L_Intrusion_Event_Count;
            ELSE
                L_Combined_First_Event_MS := VI_System_Time_MS;
                L_Combined_Event_Count := L_Intrusion_Event_Count;
            END_IF;
        END_IF;
    END_IF;

    IF L_Combined_Window_Active THEN
        IF VI_System_Time_MS >= L_Combined_First_Event_MS THEN
            L_Combined_Elapsed_MS := VI_System_Time_MS - L_Combined_First_Event_MS;
        ELSE
            L_Combined_Elapsed_MS := (4294967295 - L_Combined_First_Event_MS) + VI_System_Time_MS + 1;
        END_IF;

        IF L_Combined_Elapsed_MS > L_Combined_Window_MS THEN
            L_Combined_Window_Active := FALSE;
            L_Combined_Event_Count := 0;
        END_IF;
    END_IF;

    IF (L_Intrusion_Active_Count >= 2) OR (L_Combined_Window_Active AND (L_Combined_Event_Count >= 2)) THEN
        VO_Alarm_Active := TRUE;
        VO_Siren_Active := TRUE;
        L_Pin_Entry_Active := FALSE;
        VO_Status_Msg := 'ТРЕВОГА! Комбинированное нарушение периметра';
    ELSIF L_Any_Sensor_Active THEN
        L_Pin_Entry_Active := TRUE;
    END_IF;

    L_Alarm_Delay_Timer(IN := L_Pin_Entry_Active, PT := TO_TIME(L_Pin_Entry_Timeout_MS), VI_System_Time_MS := VI_System_Time_MS);

    IF L_Alarm_Delay_Timer.Q THEN
        VO_Alarm_Active := TRUE;
        VO_Siren_Active := TRUE;
        VO_Status_Msg := 'ТРЕВОГА! Нарушение периметра';
    ELSIF L_Pin_Entry_Active AND NOT VO_Alarm_Active THEN
        VO_Status_Msg := 'Внимание! Введите PIN-код для отмены тревоги';
    END_IF;
ELSE
    L_Any_Sensor_Active := FALSE;
    L_Intrusion_Active_Count := 0;
    L_Intrusion_Event_Count := 0;
    L_Pin_Entry_Active := FALSE;
    L_Alarm_Delay_Timer(IN := FALSE, PT := T#0s, VI_System_Time_MS := VI_System_Time_MS);
END_IF;

GVL_SECURITY_WORKFLOW.G_Arming_In_Progress := L_Arming_In_Progress;
GVL_SECURITY_WORKFLOW.G_Arm_Delay_ET := L_Arm_Delay_Timer.ET;
GVL_SECURITY_WORKFLOW.G_Arm_Delay_Q := L_Arm_Delay_Timer.Q;
GVL_SECURITY_WORKFLOW.G_Pin_Entry_Active := L_Pin_Entry_Active;
GVL_SECURITY_WORKFLOW.G_Entry_Delay_ET := L_Alarm_Delay_Timer.ET;
GVL_SECURITY_WORKFLOW.G_Entry_Delay_Q := L_Alarm_Delay_Timer.Q;
GVL_SECURITY_WORKFLOW.G_Pin_Fail_Count := L_PIN_Fail_Count;
GVL_SECURITY_WORKFLOW.G_Max_Attempts := L_Max_Attempts;
GVL_SECURITY_WORKFLOW.G_Disarm_Pending := L_Disarm_Pending;
GVL_SECURITY_WORKFLOW.G_2FA_Required := L_2FA_Required;
GVL_SECURITY_WORKFLOW.G_2FA_Send_Code_Req := VO_Send_Code_Req;
GVL_SECURITY_WORKFLOW.G_Combined_Window_Active := L_Combined_Window_Active;
GVL_SECURITY_WORKFLOW.G_Combined_Event_Count := L_Combined_Event_Count;
GVL_SECURITY_WORKFLOW.G_Intrusion_Active_Count := L_Intrusion_Active_Count;
GVL_SECURITY_WORKFLOW.G_Intrusion_Event_Count := L_Intrusion_Event_Count;
GVL_SECURITY_WORKFLOW.G_Any_Sensor_Active := L_Any_Sensor_Active;
GVL_SECURITY_WORKFLOW.G_Door_Blocking_Open := L_Door_Blocking_Open;
GVL_SECURITY_WORKFLOW.G_Window_Blocking_Open := L_Window_Blocking_Open;
GVL_SECURITY_WORKFLOW.G_Status_Text := VO_Status_Msg;
GVL_SECURITY_WORKFLOW.G_Last_Update_MS := VI_System_Time_MS;

// >>> BULK_SYNC_ANCHOR: FB_Security_System_Manager <<<
END_FUNCTION_BLOCK

(* ---- FB_Sensor_Calibration.st ---- *)
FUNCTION_BLOCK FB_Sensor_Calibration
VAR_INPUT
    VI_Sensor_ID : UDINT;
    VI_Reference_Value : REAL;
    VI_Current_Value : REAL;
    VI_Apply : BOOL;
END_VAR
VAR_OUTPUT
    VO_Offset : REAL;
    VO_Multiplier : REAL := 1.0;
    VO_Done : BOOL;
END_VAR
VAR
    L_Applied : BOOL;
END_VAR

IF VI_Apply AND NOT L_Applied THEN
    // Простая калибровка смещением (одноточечная)
    VO_Offset := VI_Reference_Value - VI_Current_Value;
    VO_Done := TRUE;
    L_Applied := TRUE;
ELSIF NOT VI_Apply THEN
    VO_Done := FALSE;
    L_Applied := FALSE;
END_IF;
END_FUNCTION_BLOCK

(* ---- FB_Sensor_Calibration_Processor.st ---- *)
FUNCTION_BLOCK FB_Sensor_Calibration_Processor
VAR_INPUT
    VI_Raw_Value : REAL;
    VI_Record    : ST_Sensor_Calibration_Record;
END_VAR
VAR_OUTPUT
    VO_Calibrated_Value : REAL;
END_VAR

VO_Calibrated_Value := (VI_Raw_Value * VI_Record.multiplier) + VI_Record.offset;

(* ---- FB_Simulation_Manager.st ---- *)
FUNCTION_BLOCK FB_Simulation_Manager
VAR_INPUT
    VI_System_Time_MS : UDINT; // Системное время (мс)
    VI_IsActivePLC    : BOOL; // Флаг: Данный ПЛК является ведущим
    VI_Scenario       : E_SCENARIO_TYPE; // Текущий активный сценарий
    VI_Config         : ST_Scenario_Config; // Конфигурация сценариев
END_VAR
VAR_OUTPUT
    VO_Sim_Lights     : ARRAY[1..32] OF BOOL; // Симулированные сигналы включения света
    VO_Sim_Active     : BOOL; // Флаг: Симуляция присутствия активна
    // Симуляция аварий (для тестирования)
    VO_Sim_Water_Leak : ARRAY[1..GVL_CONSTANTS.C_MAX_FLOOD_SENSORS] OF BOOL; // Симулированные сигналы протечки
    VO_Sim_Gas_Leak   : ARRAY[1..GVL_CONSTANTS.C_MAX_METHANE_SENSORS] OF REAL; // Симулированные уровни газа
END_VAR
VAR
    L_Random          : FB_Random_Generator;
    L_Last_Toggle     : UDINT;
    L_i               : INT;
    L_Rand_Val        : UDINT;
    L_Test_Mode       : BOOL := FALSE; // Флаг тестового режима
END_VAR

IF VI_Scenario = E_SCENARIO_TYPE.SCENARIO_AWAY AND VI_Config.Presence_Simulation_Enabled THEN
    VO_Sim_Active := TRUE;

    // Переключаем свет каждые 30 минут
    IF (VI_System_Time_MS - L_Last_Toggle) >= (GVL_CONSTANTS.C_MS_IN_MINUTE * 30) THEN
        L_Last_Toggle := VI_System_Time_MS;

        FOR L_i := 1 TO 32 DO
            L_Rand_Val := 1;
            VO_Sim_Lights[L_i] := (L_Rand_Val > 80); // 20% шанс включения
        END_FOR;
    END_IF;
ELSE
    VO_Sim_Active := FALSE;
    FOR L_i := 1 TO 32 DO VO_Sim_Lights[L_i] := FALSE; END_FOR;
END_IF;

// Симуляция аварий в тестовом режиме
IF L_Test_Mode THEN
    // Генерация случайных протечек (очень редко)
    L_Rand_Val := 1;
    IF L_Rand_Val = 42 THEN
        VO_Sim_Water_Leak[1] := TRUE;
    END_IF;

    // Симуляция утечки газа
    L_Rand_Val := 1;
    IF L_Rand_Val = 77 THEN
        VO_Sim_Gas_Leak[1] := 15.0; // 15% LEL
    END_IF;
ELSE
    FOR L_i := 1 TO GVL_CONSTANTS.C_MAX_FLOOD_SENSORS DO VO_Sim_Water_Leak[L_i] := FALSE; END_FOR;
    FOR L_i := 1 TO GVL_CONSTANTS.C_MAX_METHANE_SENSORS DO VO_Sim_Gas_Leak[L_i] := 0.0; END_FOR;
END_IF;
// >>> BULK_SYNC_ANCHOR: FB_Simulation_Manager <<<

(* ---- FB_Smoke_Detector.st ---- *)
FUNCTION_BLOCK FB_Smoke_Detector
VAR_INPUT
    VI_Smoke_Signal : BOOL;
END_VAR
VAR_OUTPUT
    VO_Smoke_Detected : BOOL;
END_VAR

VO_Smoke_Detected := VI_Smoke_Signal;

(* ---- FB_Socket_Manager.st ---- *)
FUNCTION_BLOCK FB_Socket_Manager
VAR_INPUT
    VI_System_Time_MS : UDINT;
    VI_IsActivePLC : BOOL;
    VI_Scenario : E_SCENARIO_TYPE;
    VI_Fire_Alarm : BOOL;
    VI_Flood_Alarm : BOOL;
    VI_Security_Armed : BOOL;
END_VAR
VAR_IN_OUT
    VI_Manual_Override : ARRAY[1..GVL_CONSTANTS.C_MAX_SOCKETS] OF BOOL;
    VI_Physical_Switches : ARRAY[1..GVL_CONSTANTS.C_MAX_SOCKETS] OF BOOL;
    VI_Rule_Actions : ARRAY[1..GVL_CONSTANTS.C_MAX_RULES] OF ST_Rule_Action;
    VI_IO_Modules_Online : ARRAY[1..GVL_CONSTANTS.C_MAX_MODULES] OF BOOL;
END_VAR
VAR_OUTPUT
    VO_Socket_States : ARRAY[1..GVL_CONSTANTS.C_MAX_SOCKETS] OF BOOL;
    VO_Internal_States : ARRAY[1..GVL_CONSTANTS.C_MAX_SOCKETS] OF BOOL;
END_VAR
VAR
    L_i : INT;
    L_j : INT;
    L_Rule_State : BOOL;
    L_Rule_Active : BOOL;
    L_Internal_State : ARRAY[1..GVL_CONSTANTS.C_MAX_SOCKETS] OF BOOL;
    L_Manual_Trig : ARRAY[1..GVL_CONSTANTS.C_MAX_SOCKETS] OF R_TRIG;
END_VAR

FOR L_i := 1 TO GVL_CONSTANTS.C_MAX_SOCKETS DO
    VO_Socket_States[L_i] := FALSE;
    VO_Internal_States[L_i] := L_Internal_State[L_i];
END_FOR;

IF NOT VI_IsActivePLC THEN
    RETURN;
END_IF;

FOR L_i := 1 TO GVL_CONSTANTS.C_MAX_MODULES DO
    IF NOT VI_IO_Modules_Online[L_i] THEN
        RETURN;
    END_IF;
END_FOR;

FOR L_i := 1 TO GVL_CONSTANTS.C_MAX_SOCKETS DO
    L_Rule_Active := FALSE;
    L_Rule_State := FALSE;

    L_Manual_Trig[L_i](CLK := VI_Manual_Override[L_i]);

    IF L_Manual_Trig[L_i].Q THEN
        L_Internal_State[L_i] := NOT L_Internal_State[L_i];
    END_IF;

    FOR L_j := 1 TO GVL_CONSTANTS.C_MAX_RULES DO
        IF VI_Rule_Actions[L_j].Active AND VI_Rule_Actions[L_j].Target_ID = L_i THEN
            IF VI_Rule_Actions[L_j].Action_Type = E_Rule_Action_Type.ACTION_SET_SOCKET THEN
                L_Rule_Active := TRUE;
                L_Rule_State := (VI_Rule_Actions[L_j].Value > 0.5);
                L_Internal_State[L_i] := L_Rule_State;
            ELSIF VI_Rule_Actions[L_j].Action_Type = E_Rule_Action_Type.ACTION_TOGGLE_SOCKET AND VI_Rule_Actions[L_j].Triggered THEN
                L_Internal_State[L_i] := NOT L_Internal_State[L_i];
            END_IF;
        END_IF;
    END_FOR;

    IF VI_Fire_Alarm OR VI_Flood_Alarm THEN
        IF L_i > 4 THEN
            VO_Socket_States[L_i] := FALSE;
        ELSE
            VO_Socket_States[L_i] := L_Internal_State[L_i];
        END_IF;
    ELSIF VI_Scenario = E_SCENARIO_TYPE.SCENARIO_AWAY OR VI_Security_Armed THEN
        IF L_i > 4 THEN
            VO_Socket_States[L_i] := FALSE;
        ELSE
            VO_Socket_States[L_i] := L_Internal_State[L_i];
        END_IF;
    ELSE
        IF L_Rule_Active THEN
            VO_Socket_States[L_i] := L_Rule_State;
        ELSE
            VO_Socket_States[L_i] := L_Internal_State[L_i];
        END_IF;
    END_IF;
END_FOR;

VO_Internal_States := L_Internal_State;

END_FUNCTION_BLOCK
// >>> BULK_SYNC_ANCHOR: FB_Socket_Manager <<<

(* ---- FB_Socket_V2_Staging.st ---- *)
FUNCTION_BLOCK FB_Socket_V2_Staging
VAR_INPUT
    VI_Socket_ID : INT;
    VI_Enable : BOOL;
    VI_Target_State : BOOL;
    VI_Manual_Override : BOOL;
    VI_Safety_Lock : BOOL;
    VI_Scenario_ID : INT;
    VI_Is_On : BOOL;
    VI_Manual_Override_Active : BOOL;
    VI_Safety_Blocked : BOOL;
    VI_Alarm_Active : BOOL;
END_VAR
VAR_OUTPUT
    VO_Command_Shadow : ST_Socket_Command_V2;
    VO_State_Shadow : ST_Socket_State_V2;
END_VAR

VO_Command_Shadow.Target_State := VI_Target_State;
VO_State_Shadow.Is_On := VI_Is_On;
VO_State_Shadow.Safety_Blocked := VI_Safety_Blocked;
END_FUNCTION_BLOCK

(* ---- FB_State_Manager.st ---- *)
FUNCTION_BLOCK FB_State_Manager
VAR_INPUT
    VI_System_Severity : E_System_Severity;
    VI_Root_Cause      : E_System_Root_Cause;
    VI_Freeze_Risk     : BOOL := FALSE;
END_VAR

VAR_OUTPUT
    VO_System_OK        : BOOL;
    VO_System_Warning   : BOOL;
    VO_System_Critical  : BOOL;
    VO_Status_Msg       : STRING(200);

    // compatibility output for existing orchestration
    VO_System_Mode      : E_System_Operating_Mode;
END_VAR

VO_System_OK := FALSE;
VO_System_Warning := FALSE;
VO_System_Critical := FALSE;
VO_Status_Msg := '';
VO_System_Mode := E_System_Operating_Mode.MODE_NORMAL;

CASE VI_System_Severity OF
    E_System_Severity.SEV_NORMAL:
        VO_System_OK := TRUE;
        VO_Status_Msg := 'Система в норме';
        VO_System_Mode := E_System_Operating_Mode.MODE_NORMAL;

    E_System_Severity.SEV_WARNING:
        VO_System_Warning := TRUE;
        VO_System_Mode := E_System_Operating_Mode.MODE_DEGRADED;
        CASE VI_Root_Cause OF
            E_System_Root_Cause.ROOT_WATER_LEAK:
                VO_Status_Msg := 'Предупреждение: протечка воды';
            E_System_Root_Cause.ROOT_CO_WARNING:
                VO_Status_Msg := 'Предупреждение: повышенный CO';
            ELSE
                VO_Status_Msg := 'Предупреждение системы';
        END_CASE;

    E_System_Severity.SEV_DEGRADED:
        VO_System_Warning := TRUE;
        VO_System_Mode := E_System_Operating_Mode.MODE_DEGRADED;
        CASE VI_Root_Cause OF
            E_System_Root_Cause.ROOT_SENSOR_FAULT:
                VO_Status_Msg := 'Деградация: ошибка датчика';
            E_System_Root_Cause.ROOT_IO_OFFLINE:
                VO_Status_Msg := 'Деградация: модуль IO недоступен';
            E_System_Root_Cause.ROOT_COMM_FAULT:
                VO_Status_Msg := 'Деградация: ошибка связи';
            E_System_Root_Cause.ROOT_WATCHDOG_FAULT:
                VO_Status_Msg := 'Деградация: watchdog fault';
            E_System_Root_Cause.ROOT_SUBSYSTEM_FAULT:
                VO_Status_Msg := 'Деградация: ошибка подсистемы';
            ELSE
                VO_Status_Msg := 'Деградация системы';
        END_CASE;

    E_System_Severity.SEV_CRITICAL:
        VO_System_Critical := TRUE;

        IF (VI_Root_Cause = E_System_Root_Cause.ROOT_GAS_LEAK OR
            VI_Root_Cause = E_System_Root_Cause.ROOT_CO_CRITICAL) AND
            VI_Freeze_Risk THEN
            VO_System_Mode := E_System_Operating_Mode.MODE_FREEZE_PROTECTION;
        ELSE
            VO_System_Mode := E_System_Operating_Mode.MODE_SAFE_STOP;
        END_IF;

        CASE VI_Root_Cause OF
            E_System_Root_Cause.ROOT_FIRE:
                VO_Status_Msg := 'АВАРИЯ: ПОЖАР';
            E_System_Root_Cause.ROOT_GAS_LEAK:
                VO_Status_Msg := 'АВАРИЯ: УТЕЧКА ГАЗА';
            E_System_Root_Cause.ROOT_CO_CRITICAL:
                VO_Status_Msg := 'АВАРИЯ: КРИТИЧЕСКИЙ CO';
            E_System_Root_Cause.ROOT_WATCHDOG_FAULT:
                VO_Status_Msg := 'АВАРИЯ: WATCHDOG';
            ELSE
                VO_Status_Msg := 'АВАРИЯ СИСТЕМЫ';
        END_CASE;
END_CASE;
// >>> BULK_SYNC_ANCHOR: FB_State_Manager <<<

(* ---- FB_State_Replication.st ---- *)
FUNCTION_BLOCK FB_State_Replication
VAR_INPUT
    VI_Local_Role : E_PLC_ROLE; // Локальная роль ПЛК (Active/Standby)
    VI_Sync_Req : BOOL; // Запрос на принудительную синхронизацию
    VI_Local_State : ST_System_State_Snapshot; // Локальное состояние системы
    VI_Remote_State : ST_System_State_Snapshot; // Состояние системы партнера
    VI_System_Time_MS : UDINT; // Системное время (мс)
END_VAR
VAR_OUTPUT
    VO_State_Updated : BOOL; // Флаг: Состояние было обновлено
    VO_Synced_State : ST_System_State_Snapshot; // Синхронизированное состояние
END_VAR
VAR
    L_Sync_In_Progress : BOOL;
    L_Last_Sync_Time : UDINT;
    L_Periodic_Sync_Req : BOOL;
    L_Elapsed_Time : UDINT;
END_VAR

// Периодическая синхронизация (каждые 5 секунд)
L_Elapsed_Time := (SEL(VI_System_Time_MS >= L_Last_Sync_Time, VI_System_Time_MS - L_Last_Sync_Time, (4294967295 - L_Last_Sync_Time) + VI_System_Time_MS + 1));

IF L_Elapsed_Time > 5000 THEN
    L_Periodic_Sync_Req := TRUE;
    L_Last_Sync_Time := VI_System_Time_MS;
ELSE
    L_Periodic_Sync_Req := FALSE;
END_IF;

// State Replication Logic
// Синхронизация состояния между ПЛК (ТЗ 8.2)
IF (VI_Sync_Req OR L_Periodic_Sync_Req) AND NOT L_Sync_In_Progress THEN
    L_Sync_In_Progress := TRUE;

    // Разрешение конфликтов на основе версии состояния
    IF VI_Remote_State.Version > VI_Local_State.Version THEN
        VO_Synced_State := VI_Remote_State;
        VO_State_Updated := TRUE;
    ELSIF VI_Remote_State.Version = VI_Local_State.Version THEN
        // Если версии равны, приоритет у ведущего ПЛК
        IF VI_Local_Role = E_PLC_ROLE.ROLE_STANDBY THEN
            VO_Synced_State := VI_Remote_State;
            VO_State_Updated := TRUE;
        ELSE
            VO_Synced_State := VI_Local_State;
            VO_State_Updated := FALSE;
        END_IF;
    ELSE
        VO_Synced_State := VI_Local_State;
        VO_State_Updated := FALSE;
    END_IF;
ELSIF NOT (VI_Sync_Req OR L_Periodic_Sync_Req) THEN
    L_Sync_In_Progress := FALSE;
    VO_State_Updated := FALSE;
    VO_Synced_State := VI_Local_State;
END_IF;

(* ---- FB_State_Snapshot_Manager.st ---- *)
FUNCTION_BLOCK FB_State_Snapshot_Manager
VAR_INPUT
    VI_System_Time_MS : UDINT;
    VI_Trigger_Event  : BOOL; // Сигнал на создание снимка
    VI_Event_Code     : WORD;
    VI_Current_State  : ST_State_Snapshot;
END_VAR
VAR_OUTPUT
    VO_Snapshot_Saved : BOOL;
END_VAR
VAR
    L_Snapshot_Buffer : ARRAY[1..GVL_CONSTANTS.C_MAX_STATE_SNAPSHOTS] OF ST_State_Snapshot;
    L_Write_Idx       : INT := 1;
END_VAR

IF VI_Trigger_Event THEN
    L_Snapshot_Buffer[L_Write_Idx] := VI_Current_State;
    L_Snapshot_Buffer[L_Write_Idx].timestamp_ms := VI_System_Time_MS;

    // NOTE:
    // ST_State_Snapshot no longer contains trigger_event_code in live project.
    // VI_Event_Code is reserved for future snapshot metadata extension.

    L_Write_Idx := (L_Write_Idx MOD GVL_CONSTANTS.C_MAX_STATE_SNAPSHOTS) + 1;
    VO_Snapshot_Saved := TRUE;
ELSE
    VO_Snapshot_Saved := FALSE;
END_IF;

(* ---- FB_State_Trace_Log.st ---- *)
FUNCTION_BLOCK FB_State_Trace_Log
VAR_INPUT
    VI_System_Time : UDINT;
    VI_Gas_Alarm : BOOL;
    VI_Leak_Alarm : BOOL;
    VI_Pumps : ARRAY[1..GVL_CONSTANTS.C_MAX_MANIFOLDS] OF BOOL;
END_VAR
VAR_OUTPUT
    VO_Last_Change_Time : UDINT;
END_VAR
VAR
    L_Last_Gas : BOOL;
    L_Last_Leak : BOOL;
END_VAR

IF (VI_Gas_Alarm <> L_Last_Gas) OR (VI_Leak_Alarm <> L_Last_Leak) THEN
    VO_Last_Change_Time := VI_System_Time;
END_IF;

L_Last_Gas := VI_Gas_Alarm;
L_Last_Leak := VI_Leak_Alarm;
END_FUNCTION_BLOCK

(* ---- FB_System_Alarm_Orchestrator.st ---- *)
// ==============================================================================
// System alarm orchestrator helper
//
// Internal helper for PRG_System.
// Owns FB_Alarm_Manager call and alarm output projection.
// ==============================================================================
FUNCTION_BLOCK FB_System_Alarm_Orchestrator
VAR_INPUT
    VI_First_Fault_Active : BOOL;
    VI_First_Fault_Type : INT;
    VI_First_Fault_Source : INT;
END_VAR

VAR
    fbAlarmManager : FB_Alarm_Manager;
END_VAR

fbAlarmManager(
    VI_System_Time_MS := GVL_STATUS.G_System_Time_MS,
    VI_IsActivePLC := GVL_STATUS.G_Is_Active_PLC,
    VI_Gas_Alarm := GVL_HEALTH_BRIDGE.G_Gas_Detected OR GVL_HEALTH_BRIDGE.G_CO_Alarm_Level,
    VI_Fire_Alarm := GVL_HEALTH_BRIDGE.G_Smoke_Detected,
    VI_Flood_Alarm := GVL_HEALTH_BRIDGE.G_Leak_Detected,
    VI_Security_Alarm := GVL_ALARM.G_Security_Alarm,
    VI_First_Fault_Active := VI_First_Fault_Active,
    VI_First_Fault_Type := VI_First_Fault_Type,
    VI_First_Fault_Source := VI_First_Fault_Source,
    VI_Boiler_Errors := GVL_STATE.G_Boiler_Error,
    VI_Security_Msg := GVL_STATUS.G_Security_Status_Msg,
    VI_Acknowledge_All := GVL_CONFIG.G_HMI_Ack_Alarms OR GVL_COMMAND.G_Reset_Errors,
    VI_Mute_Siren := GVL_ALARM_AUDIBLE_ACK.G_Ack_Active,
    VIO_Next_Alarm_ID := GVL_ALARM.G_Next_Alarm_ID,
    VO_Global_Critical => GVL_ALARM.G_Global_Critical,
    VO_Global_Warning => GVL_ALARM.G_Global_Warning,
    VO_Siren_Active => GVL_ALARM.G_Global_Siren,
    VO_Active_Count => GVL_ALARM.G_Active_Alarm_Count,
    VO_Unacked_Count => GVL_ALARM.G_Unacked_Alarm_Count,
    VO_Event_Pulse => GVL_STATUS.G_Diagnostics.Alarm_Event_Pulse,
    VO_Event_Code => GVL_STATUS.G_Diagnostics.Alarm_Event_Code,
    VO_Event_Value => GVL_STATUS.G_Diagnostics.Alarm_Event_Value,
    VO_Alarm_List => GVL_ALARM.G_Alarm_List
);

// >>> BULK_SYNC_ANCHOR: FB_System_Alarm_Orchestrator <<<
END_FUNCTION_BLOCK

(* ---- FB_System_Coordinator.st ---- *)
FUNCTION_BLOCK FB_System_Coordinator

VAR_INPUT
    VI_Fire_Latched : BOOL;
    VI_Gas_Latched : BOOL;
    VI_Leak_Latched : BOOL;

    VI_IO_Degraded : BOOL;
    VI_Ownership_Violation : BOOL;

    VI_Behavior_Mode : E_Behavior_Mode;
END_VAR

VAR_OUTPUT
    VO_Block_Heating : BOOL;
    VO_Block_Ventilation : BOOL;
    VO_Block_Lighting : BOOL;
    VO_Block_Sockets : BOOL;

    VO_System_Degraded : BOOL;

    VO_Code : UDINT;
END_VAR

// reset
VO_Block_Heating := FALSE;
VO_Block_Ventilation := FALSE;
VO_Block_Lighting := FALSE;
VO_Block_Sockets := FALSE;
VO_System_Degraded := FALSE;
VO_Code := 0;

// FIRE has highest priority. Safety-stop ownership remains in PRG_Safety.
IF VI_Fire_Latched THEN
    VO_Block_Heating := TRUE;
    VO_Block_Ventilation := TRUE;
    VO_Block_Sockets := TRUE;
    VO_Code := 100;
    RETURN;
END_IF;

// GAS has higher priority than behavior mode.
IF VI_Gas_Latched THEN
    VO_Block_Heating := TRUE;
    VO_Block_Lighting := TRUE;
    VO_Block_Sockets := TRUE;
    VO_Code := 200;
    RETURN;
END_IF;

// LEAK blocks heating but does not suppress later degradation/mode overlays.
IF VI_Leak_Latched THEN
    VO_Block_Heating := TRUE;
    VO_Code := 300;
END_IF;

// IO degraded blocks heating and marks system degraded.
IF VI_IO_Degraded THEN
    VO_System_Degraded := TRUE;
    VO_Block_Heating := TRUE;
    IF VO_Code = 0 THEN
        VO_Code := 400;
    END_IF;
END_IF;

// Ownership violation marks system degraded. Test/result handler owns any safe-stop reaction.
IF VI_Ownership_Violation THEN
    VO_System_Degraded := TRUE;
    IF VO_Code = 0 THEN
        VO_Code := 500;
    END_IF;
END_IF;

// Behavior mode overlays. These are lower priority than safety/system faults.
CASE VI_Behavior_Mode OF
    BEHAVIOR_AWAY:
        VO_Block_Lighting := TRUE;
        VO_Block_Sockets := TRUE;
        IF VO_Code = 0 THEN
            VO_Code := 600;
        END_IF;

    BEHAVIOR_NIGHT:
        VO_Block_Lighting := TRUE;
        IF VO_Code = 0 THEN
            VO_Code := 700;
        END_IF;

    BEHAVIOR_MAINTENANCE:
        VO_Block_Heating := TRUE;
        VO_Block_Ventilation := TRUE;
        IF VO_Code = 0 THEN
            VO_Code := 800;
        END_IF;
ELSE
        // No fallback required
END_CASE;
END_FUNCTION_BLOCK

(* ---- FB_System_Diagnostics_Publisher.st ---- *)
FUNCTION_BLOCK FB_System_Diagnostics_Publisher
VAR_INPUT
    VI_Enable : BOOL;
    VI_System_Time_MS : UDINT;
    VI_Backup_Pump_Out_Of_Service : BOOL;
    VI_Electric_Heater_Out_Of_Service : BOOL;
    VI_Manifold_Pump_Out_Of_Service : ARRAY[1..GVL_CONSTANTS.C_MAX_MANIFOLDS] OF BOOL;
    VI_DHW_Heating_Pump_Out_Of_Service : BOOL;
    VI_DHW_Circ_Pump_Out_Of_Service : BOOL;
    VI_User_Access_Level : INT;
    VI_Dangerous_Action_Pending : BOOL;
    VI_Dangerous_Action_Text : STRING(160);
    VI_Sensor_Fault : BOOL;
    VI_IO_Offline : BOOL;
    VI_Subsystem_Degraded : BOOL;
    VI_Manifold_Pressure_Fault : ARRAY[1..GVL_CONSTANTS.C_MAX_MANIFOLDS] OF BOOL;
    VI_Manifold_Current_Fault : ARRAY[1..GVL_CONSTANTS.C_MAX_MANIFOLDS] OF BOOL;
    VI_Manifold_Return_Temp_Fault : ARRAY[1..GVL_CONSTANTS.C_MAX_MANIFOLDS] OF BOOL;
END_VAR
VAR_OUTPUT
    VO_Diagnostics : ST_System_Diagnostics;
    VO_Publication_Valid : BOOL;
    VO_Status_Code : UINT;
    VO_Status_Text : STRING(128);
END_VAR
VAR
    L_i : INT;
    L_Pressure_First : INT;
    L_Current_First : INT;
    L_Return_First : INT;
    L_Any_Manifold_Fault : BOOL;
END_VAR

VO_Diagnostics.Freeze_Hardware_Event_Pending := FALSE;
VO_Diagnostics.Freeze_Hardware_Event_Text := '';
VO_Diagnostics.Backup_Pump_Fault := VI_Backup_Pump_Out_Of_Service;
VO_Diagnostics.Electric_Heater_Fault := VI_Electric_Heater_Out_Of_Service;
VO_Diagnostics.Backup_Pump_Recovered_After_Retry := FALSE;
VO_Diagnostics.Electric_Heater_Recovered_After_Retry := FALSE;
VO_Diagnostics.Backup_Pump_Out_Of_Service := VI_Backup_Pump_Out_Of_Service;
VO_Diagnostics.Electric_Heater_Out_Of_Service := VI_Electric_Heater_Out_Of_Service;

VO_Diagnostics.Pump_Exercise_Active := FALSE;
VO_Diagnostics.Pump_Exercise_Failed := FALSE;
VO_Diagnostics.Pump_Exercise_Last_Equipment := '';
VO_Diagnostics.Pump_Exercise_Last_Result := 'Pump exercise publisher passive';
VO_Diagnostics.Pump_Exercise_No_Feedback_Count := 0;
VO_Diagnostics.DHW_Heating_Pump_Exercise_Count := 0;
VO_Diagnostics.DHW_Circ_Pump_Exercise_Count := 0;
VO_Diagnostics.Backup_Pump_Exercise_Count := 0;
VO_Diagnostics.Pump_Exercise_Event_Seq := VI_System_Time_MS;
VO_Diagnostics.Pump_Exercise_Journal_1 := 'Passive diagnostics publication active';
VO_Diagnostics.Pump_Exercise_Journal_2 := '';
VO_Diagnostics.Pump_Exercise_Journal_3 := '';
VO_Diagnostics.Pump_Exercise_Journal_Last_Seq := VI_System_Time_MS;

VO_Diagnostics.Pump_Maintenance_Required := VI_Backup_Pump_Out_Of_Service OR VI_Electric_Heater_Out_Of_Service;
VO_Diagnostics.Pump_Maintenance_Warning := VO_Diagnostics.Pump_Maintenance_Required;

VO_Diagnostics.DHW_Heating_Pump_Out_Of_Service := VI_DHW_Heating_Pump_Out_Of_Service;
VO_Diagnostics.DHW_Circ_Pump_Out_Of_Service := VI_DHW_Circ_Pump_Out_Of_Service;

VO_Diagnostics.Maintenance_Last_Action := 'Diagnostics publication only';
VO_Diagnostics.Operator_Action_Blocked := FALSE;
VO_Diagnostics.Operator_Block_Reason := '';
VO_Diagnostics.Operator_Last_Forbidden_Action := '';
VO_Diagnostics.Operator_Journal_1 := 'Operator diagnostics passive';
VO_Diagnostics.Operator_Journal_2 := '';
VO_Diagnostics.Operator_Journal_3 := '';
VO_Diagnostics.Operator_Journal_Event_Seq := VI_System_Time_MS;
VO_Diagnostics.Operator_Journal_Last_Seq := VI_System_Time_MS;

VO_Diagnostics.Dangerous_Action_Pending_Confirm := VI_Dangerous_Action_Pending;
VO_Diagnostics.Dangerous_Action_Confirm_Text := VI_Dangerous_Action_Text;
VO_Diagnostics.Dangerous_Action_Confirm_Deadline_MS := 0;
VO_Diagnostics.User_Access_Level_Active := VI_User_Access_Level;
VO_Diagnostics.User_Access_Denied := FALSE;
VO_Diagnostics.User_Access_Deny_Reason := '';

VO_Diagnostics.Valve_Test_Mode_Active := FALSE;
VO_Diagnostics.Valve_Test_Deadline_MS := 0;
VO_Diagnostics.Valve_Test_Remaining_MS := 0;
VO_Diagnostics.Valve_Test_Validation_OK := TRUE;
VO_Diagnostics.Valve_Test_Validation_Text := 'No generic valve test active';
VO_Diagnostics.Valve_Test_Forced_Close := FALSE;

VO_Diagnostics.Water_Valve_Test_Mode_Active := FALSE;
VO_Diagnostics.Water_Valve_Test_Deadline_MS := 0;
VO_Diagnostics.Water_Valve_Test_Remaining_MS := 0;
VO_Diagnostics.Water_Valve_Test_Validation_OK := TRUE;
VO_Diagnostics.Water_Valve_Test_Validation_Text := 'No water valve test active';
VO_Diagnostics.Water_Valve_Test_Forced_Close := FALSE;
VO_Diagnostics.Gas_Valve_Test_Mode_Active := FALSE;
VO_Diagnostics.Gas_Valve_Test_Deadline_MS := 0;
VO_Diagnostics.Gas_Valve_Test_Remaining_MS := 0;
VO_Diagnostics.Gas_Valve_Test_Validation_OK := TRUE;
VO_Diagnostics.Gas_Valve_Test_Validation_Text := 'No gas valve test active';
VO_Diagnostics.Gas_Valve_Test_Forced_Close := FALSE;

VO_Diagnostics.Active_Leak_Sensor_Index := 0;
VO_Diagnostics.Active_Gas_Sensor_Index := 0;
VO_Diagnostics.Active_Leak_Zone_Name := '';
VO_Diagnostics.Active_Gas_Zone_Name := '';
VO_Diagnostics.Water_Valve_Test_Context := 'Water diagnostics passive';
VO_Diagnostics.Gas_Valve_Test_Context := 'Gas diagnostics passive';

VO_Diagnostics.Water_Recovery_Target_Zone_Index := 0;
VO_Diagnostics.Gas_Recovery_Target_Zone_Index := 0;
VO_Diagnostics.Water_Recovery_Selective_Allowed := FALSE;
VO_Diagnostics.Gas_Recovery_Selective_Allowed := FALSE;
VO_Diagnostics.Water_Recovery_Selective_Text := 'Selective water recovery inactive';
VO_Diagnostics.Gas_Recovery_Selective_Text := 'Selective gas recovery inactive';
VO_Diagnostics.Water_Recovery_Physical_Active := FALSE;
VO_Diagnostics.Water_Recovery_Physical_Zone_Name := '';

VO_Diagnostics.Water_Valve_Exercise_Last_Zone := 0;
VO_Diagnostics.Water_Valve_Exercise_Last_Result := 'Water valve exercise inactive';
VO_Diagnostics.Water_Close_Fault_Active := FALSE;
VO_Diagnostics.Water_Close_Fault_Zone_Name := '';
VO_Diagnostics.Water_Close_Fault_Text := '';
VO_Diagnostics.Water_Localization_Failed := FALSE;
VO_Diagnostics.Water_Main_Shutdown_Recommended := FALSE;
VO_Diagnostics.Water_Escalation_Text := '';
VO_Diagnostics.Alarm_Event_Pulse := FALSE;
VO_Diagnostics.Alarm_Event_Code := 0;
VO_Diagnostics.Alarm_Event_Value := 0.0;
VO_Diagnostics.Sensor_Fault := VI_Sensor_Fault;
VO_Diagnostics.IO_Offline := VI_IO_Offline;
VO_Diagnostics.Subsystem_Degraded := VI_Subsystem_Degraded;

L_Pressure_First := 0;
L_Current_First := 0;
L_Return_First := 0;
L_Any_Manifold_Fault := FALSE;

FOR L_i := 1 TO GVL_CONSTANTS.C_MAX_MANIFOLDS DO
    VO_Diagnostics.Manifold_Pump_Out_Of_Service[L_i] := VI_Manifold_Pump_Out_Of_Service[L_i];
    VO_Diagnostics.Manifold_Pump_Exercise_Count[L_i] := 0;

    VO_Diagnostics.Manifold_Pressure_Fault[L_i] := VI_Manifold_Pressure_Fault[L_i];
    VO_Diagnostics.Manifold_Pressure_Diag_Code[L_i] := SEL(VI_Manifold_Pressure_Fault[L_i], WORD#0, WORD#16#E004);
    IF VI_Manifold_Pressure_Fault[L_i] AND (L_Pressure_First = 0) THEN
        L_Pressure_First := L_i;
    END_IF;

    VO_Diagnostics.Manifold_Current_Fault[L_i] := VI_Manifold_Current_Fault[L_i];
    VO_Diagnostics.Manifold_Current_Diag_Code[L_i] := SEL(VI_Manifold_Current_Fault[L_i], WORD#0, WORD#16#E00A);
    IF VI_Manifold_Current_Fault[L_i] AND (L_Current_First = 0) THEN
        L_Current_First := L_i;
    END_IF;

    VO_Diagnostics.Manifold_Return_Temp_Fault[L_i] := VI_Manifold_Return_Temp_Fault[L_i];
    VO_Diagnostics.Manifold_Return_Temp_Diag_Code[L_i] := SEL(VI_Manifold_Return_Temp_Fault[L_i], WORD#0, WORD#16#E00D);
    IF VI_Manifold_Return_Temp_Fault[L_i] AND (L_Return_First = 0) THEN
        L_Return_First := L_i;
    END_IF;

    VO_Diagnostics.Manifold_Sensor_Fault_Count[L_i] := 0;
    IF VI_Manifold_Pressure_Fault[L_i] THEN
        VO_Diagnostics.Manifold_Sensor_Fault_Count[L_i] := VO_Diagnostics.Manifold_Sensor_Fault_Count[L_i] + 1;
    END_IF;
    IF VI_Manifold_Current_Fault[L_i] THEN
        VO_Diagnostics.Manifold_Sensor_Fault_Count[L_i] := VO_Diagnostics.Manifold_Sensor_Fault_Count[L_i] + 1;
    END_IF;
    IF VI_Manifold_Return_Temp_Fault[L_i] THEN
        VO_Diagnostics.Manifold_Sensor_Fault_Count[L_i] := VO_Diagnostics.Manifold_Sensor_Fault_Count[L_i] + 1;
    END_IF;

    VO_Diagnostics.Manifold_Sensor_Out_Of_Service[L_i] := VO_Diagnostics.Manifold_Sensor_Fault_Count[L_i] > 0;
    L_Any_Manifold_Fault := L_Any_Manifold_Fault OR VO_Diagnostics.Manifold_Sensor_Out_Of_Service[L_i];
END_FOR;

FOR L_i := 1 TO 32 DO
    VO_Diagnostics.Water_Zone_Open_Fault[L_i] := FALSE;
    VO_Diagnostics.Water_Zone_Close_Fault[L_i] := FALSE;
    VO_Diagnostics.Water_Zone_Critical_Close_Fault[L_i] := FALSE;
    VO_Diagnostics.Water_Zone_Close_Retry_Active[L_i] := FALSE;
    VO_Diagnostics.Water_Zone_Close_Retry_Count[L_i] := 0;
    VO_Diagnostics.Water_Zone_Close_Recovered_After_Retry[L_i] := FALSE;
END_FOR;

VO_Diagnostics.Manifold_Pressure_Fault_Active := L_Pressure_First > 0;
VO_Diagnostics.Manifold_Pressure_First_Fault_Index := L_Pressure_First;
VO_Diagnostics.Manifold_Pressure_Fault_Text := SEL(L_Pressure_First > 0, '', 'Manifold pressure fault active');

VO_Diagnostics.Manifold_Current_Fault_Active := L_Current_First > 0;
VO_Diagnostics.Manifold_Current_First_Fault_Index := L_Current_First;
VO_Diagnostics.Manifold_Current_Fault_Text := SEL(L_Current_First > 0, '', 'Manifold current fault active');

VO_Diagnostics.Manifold_Return_Temp_Fault_Active := L_Return_First > 0;
VO_Diagnostics.Manifold_Return_Temp_First_Fault_Index := L_Return_First;
VO_Diagnostics.Manifold_Return_Temp_Fault_Text := SEL(L_Return_First > 0, '', 'Manifold return temperature fault active');

VO_Diagnostics.Manifold_Sensor_Out_Of_Service_Active := L_Any_Manifold_Fault;
VO_Diagnostics.Manifold_Sensor_First_OOS_Index := SEL(L_Pressure_First > 0, SEL(L_Current_First > 0, L_Return_First, L_Current_First), L_Pressure_First);
VO_Diagnostics.Manifold_Sensor_OOS_Text := SEL(L_Any_Manifold_Fault, '', 'Manifold sensor out of service');

VO_Publication_Valid := VI_Enable;
IF VI_Subsystem_Degraded OR VI_IO_Offline OR VI_Sensor_Fault OR L_Any_Manifold_Fault THEN
    VO_Status_Code := 1;
    VO_Status_Text := 'System diagnostics degraded';
ELSE
    VO_Status_Code := 0;
    VO_Status_Text := 'System diagnostics nominal';
END_IF;

END_FUNCTION_BLOCK
// >>> BULK_SYNC_ANCHOR: FB_System_Diagnostics_Publisher <<<

(* ---- FB_System_Evacuation.st ---- *)
// ==============================================================================
// System evacuation helper
//
// Internal helper for PRG_System.
// Owns evacuation guidance logic and zone targeting.
// ==============================================================================
FUNCTION_BLOCK FB_System_Evacuation
VAR
    L_i : INT;
END_VAR

FOR L_i := 1 TO 32 DO
    IF GVL_STATE.G_Evacuation_Active[L_i] THEN
        GVL_STATE.G_Evac_Guidance[L_i] := TRUE;
        GVL_STATE.G_Evac_Target_Zone_Name[L_i] := GVL_STATE.G_Zone_Names[L_i];
    ELSE
        GVL_STATE.G_Evac_Guidance[L_i] := FALSE;
        GVL_STATE.G_Evac_Target_Zone_Name[L_i] := '';
    END_IF;
END_FOR;

// >>> BULK_SYNC_ANCHOR: FB_System_Evacuation <<<

(* ---- FB_System_Gateway_Intent.st ---- *)
FUNCTION_BLOCK FB_System_Gateway_Intent
VAR_INPUT
    VI_System_Time_MS : UDINT;
    VI_IsActivePLC : BOOL;
    VI_Gateway_Writes_Allowed : BOOL;
END_VAR

VAR_IN_OUT
    VIO_FloorHeating_Temps : ARRAY[1..GVL_CONSTANTS.C_MAX_HEATING_CIRCUITS] OF REAL;
    VIO_Zone_Valve_States : ARRAY[1..GVL_CONSTANTS.C_MAX_HEATING_CIRCUITS] OF BOOL;
    VIO_Lighting_Base_Levels : ARRAY[1..GVL_CONSTANTS.C_MAX_LIGHT_ZONES] OF BYTE;
    VIO_Scenario_Req_Gateway : E_SCENARIO_TYPE;
END_VAR

VAR
    fbGateway : FB_Gateway_Interface;
    L_Gateway_Flood_Alarm_Active : BOOL;
    L_Gateway_Gas_Alarm_Active : BOOL;
    L_Gateway_Fire_Alarm_Active : BOOL;
END_VAR

// Gateway telemetry must expose authoritative safety truth and latches,
// not stale alarm projection fields.
L_Gateway_Flood_Alarm_Active := GVL_HEALTH_BRIDGE.G_Leak_Detected OR GVL_STATE.G_Safety_Leak_Latched;
L_Gateway_Gas_Alarm_Active := GVL_HEALTH_BRIDGE.G_Gas_Detected OR GVL_HEALTH_BRIDGE.G_CO_Alarm_Level OR GVL_STATE.G_Safety_Gas_Latched;
L_Gateway_Fire_Alarm_Active := GVL_HEALTH_BRIDGE.G_Smoke_Detected OR GVL_STATE.G_Safety_Smoke_Latched;

VIO_Scenario_Req_Gateway := SCENARIO_NONE;

fbGateway(
    VI_System_Time_MS := VI_System_Time_MS,
    VI_Local_PLC_Role := SEL(VI_IsActivePLC, E_PLC_ROLE.ROLE_STANDBY, E_PLC_ROLE.ROLE_ACTIVE),
    VI_Incoming_Command := GVL_GATEWAY.G_Gateway_Command,
    VI_Command_Received := GVL_GATEWAY.G_Gateway_Command_Received,
    VI_FloorHeating_Temps := VIO_FloorHeating_Temps,
    VI_Room_Temps := GVL_STATE.G_Room_Temps,
    VI_Zone_Valve_States := VIO_Zone_Valve_States,
    VI_Manifold_Pressures := GVL_STATE.G_Manifold_Pressures,
    VI_Manifold_Pump_States := GVL_STATE.G_Manifold_Pumps,
    VI_Outdoor_Temp := GVL_STATE.G_Outdoor_Temp,
    VI_Security_Armed := GVL_ALARM.G_Security_Armed,
    VI_Flood_Alarm_Active := L_Gateway_Flood_Alarm_Active,
    VI_Gas_Alarm_Active := L_Gateway_Gas_Alarm_Active,
    VI_Fire_Alarm_Active := L_Gateway_Fire_Alarm_Active,
    VI_Methane_Concentration := GVL_STATE.G_Methane_Sensors[1],
    VI_Lighting_Base_Levels := VIO_Lighting_Base_Levels,
    VI_Socket_States := GVL_STATE.G_Socket_States,
    VI_Blinds_Positions := GVL_STATE.G_Blinds_Positions,
    VI_Active_Scenario := GVL_STATUS.G_Current_Scenario,
    VI_Send_2FA_Req := GVL_COMMAND.G_Send_2FA_Req,
    VI_2FA_Code := GVL_COMMAND.G_2FA_Code_Out,
    VI_Allowed_IPs := GVL_CONFIG.G_Allowed_IPs,
    VO_Telegram_Msg => GVL_GATEWAY.G_Gateway_Telegram_Msg,
    VO_Send_Telegram => GVL_GATEWAY.G_Gateway_Send_Telegram,
    VO_HMI_Status_Message => GVL_GATEWAY.G_Gateway_HMI_Status_Message,
    VO_Data_Ready => GVL_GATEWAY.G_Gateway_Data_Ready,
    VO_Modbus_Registers => GVL_GATEWAY.G_Gateway_Modbus_Registers,
    VO_Arm_Req => GVL_COMMAND.G_Arm_Req,
    VO_Disarm_Req => GVL_COMMAND.G_Disarm_Req,
    VO_PIN_Code => GVL_COMMAND.G_PIN_Code,
    VO_RFID_Tag => GVL_COMMAND.G_RFID_Tag,
    VO_2FA_Code_In => GVL_COMMAND.G_2FA_Code_In,
    VO_Lighting_Override => GVL_COMMAND.G_Lighting_Override,
    VO_Blinds_Override => GVL_COMMAND.G_Blinds_Override,
    VO_Socket_Override => GVL_COMMAND.G_Socket_Override,
    VO_Reset_Errors_Req => GVL_COMMAND.G_Reset_Errors
);

IF fbGateway.VO_Set_Scenario_Req THEN
    VIO_Scenario_Req_Gateway := fbGateway.VO_Target_Scenario;
END_IF;

GVL_INTENT_USER.I_Source_Valid := TRUE;
GVL_INTENT_USER.I_Last_Update_MS := VI_System_Time_MS;
GVL_INTENT_USER.I_Arm_Request := GVL_COMMAND.G_Arm_Req;
GVL_INTENT_USER.I_Disarm_Request := GVL_COMMAND.G_Disarm_Req;
GVL_INTENT_USER.I_PIN_Code := GVL_COMMAND.G_PIN_Code;
GVL_INTENT_USER.I_RFID_Tag := GVL_COMMAND.G_RFID_Tag;
GVL_INTENT_USER.I_2FA_Code_In := GVL_COMMAND.G_2FA_Code_In;
GVL_INTENT_USER.I_Lighting_Override_32 := GVL_COMMAND.G_Lighting_Override;
GVL_INTENT_USER.I_Blinds_Override_32 := GVL_COMMAND.G_Blinds_Override;
GVL_INTENT_USER.I_Socket_Override_32 := GVL_COMMAND.G_Socket_Override;
GVL_INTENT_USER.I_Reset_Errors := GVL_COMMAND.G_Reset_Errors;
GVL_INTENT_USER.I_Set_Temp_Req := fbGateway.VO_Set_Temp_Req;
GVL_INTENT_USER.I_Target_Zone := fbGateway.VO_Target_Zone;
GVL_INTENT_USER.I_Target_Temperature := fbGateway.VO_Target_Temp;
GVL_INTENT_USER.I_Set_Vent_Req := fbGateway.VO_Set_Vent_Req;
GVL_INTENT_USER.I_Target_Vent_Speed := fbGateway.VO_Target_Vent_Speed;
GVL_INTENT_USER.I_Set_Config_Req := fbGateway.VO_Set_Config_Req;
GVL_INTENT_USER.I_Time_Sync_Req := fbGateway.VO_Sync_Time_Req;
GVL_INTENT_USER.I_New_Time_MS := fbGateway.VO_New_Time_MS;

// >>> BULK_SYNC_ANCHOR: FB_System_Gateway_Intent <<<
END_FUNCTION_BLOCK

(* ---- FB_System_Health_Orchestrator.st ---- *)
// ==============================================================================
// System health orchestrator helper
//
// Internal helper for PRG_System.
// Owns safety latch update, watchdog, system health aggregation,
// system mode calculation, HMI/fault publication, diagnostic exports,
// and human-readable mode/cause text projection.
// ==============================================================================
FUNCTION_BLOCK FB_System_Health_Orchestrator
VAR_OUTPUT
    VO_First_Fault_Active : BOOL;
    VO_First_Fault_Type : INT;
    VO_First_Fault_Source : INT;
    VO_System_Severity : E_System_Severity;
    VO_Root_Cause : E_System_Root_Cause;
    VO_Watchdog_Fault : BOOL;
END_VAR

VAR
    fbSafety : FB_Safety_Manager;
    fbWatchdog : FB_Watchdog;
    fbSystemHealth : FB_System_Health;
    fbStateManager : FB_State_Manager;
    fbHMIInterface : FB_HMI_Interface;
    fbFaultLogger : FB_Fault_Logger;
END_VAR

fbSafety(
    VI_Gas_Alarm := GVL_STATE.G_Safety_Gas_Alarm,
    VI_Leak_Alarm := GVL_STATE.G_Safety_Leak_Alarm,
    VI_Smoke_Alarm := GVL_STATE.G_Safety_Smoke_Alarm,
    VI_Reset := GVL_COMMAND.G_Reset_Errors,
    VO_Gas_Latched => GVL_STATE.G_Safety_Gas_Latched,
    VO_Leak_Latched => GVL_STATE.G_Safety_Leak_Latched,
    VO_Smoke_Latched => GVL_STATE.G_Safety_Smoke_Latched,
    VO_Emergency_Stop => GVL_STATE.G_Safety_Emergency_Stop
);

GVL_STATE.G_Freeze_Hardware_Degraded := GVL_STATUS.G_Diagnostics.Backup_Pump_Fault OR GVL_STATUS.G_Diagnostics.Electric_Heater_Fault;
GVL_STATE.G_Freeze_Hardware_Failed := GVL_STATUS.G_Diagnostics.Backup_Pump_Fault AND GVL_STATUS.G_Diagnostics.Electric_Heater_Fault;

fbWatchdog(
    VI_System_Time_MS := GVL_STATUS.G_System_Time_MS
);

fbSystemHealth(
    VI_Smoke_Detected := GVL_HEALTH_BRIDGE.G_Smoke_Detected OR GVL_STATE.G_Safety_Smoke_Latched,
    VI_Gas_Detected := GVL_HEALTH_BRIDGE.G_Gas_Detected OR GVL_STATE.G_Safety_Gas_Latched,
    VI_CO_Warning_Level := GVL_HEALTH_BRIDGE.G_CO_Warning_Level,
    VI_CO_Alarm_Level := GVL_HEALTH_BRIDGE.G_CO_Alarm_Level,
    VI_Leak_Detected := GVL_HEALTH_BRIDGE.G_Leak_Detected OR GVL_STATE.G_Safety_Leak_Latched,
    VI_Sensor_Fault := GVL_STATE.G_Heating_Sensor_Fault OR GVL_STATE.G_DHW_Sensor_Fault OR GVL_STATUS.G_Diagnostics.Manifold_Pressure_Fault_Active OR GVL_STATUS.G_Diagnostics.Manifold_Current_Fault_Active OR GVL_STATUS.G_Diagnostics.Manifold_Return_Temp_Fault_Active,
    VI_IO_Offline := GVL_STATE.G_Heating_IO_Fault OR GVL_STATE.G_DHW_IO_Fault OR GVL_STATE.G_Ventilation_IO_Fault OR GVL_STATE.G_Lighting_IO_Fault,
    VI_Comm_Fault := GVL_STATE.G_Access_Comm_Fault,
    VI_Watchdog_Fault := fbWatchdog.VO_Watchdog_Fault,
    VI_Subsystem_Fault := GVL_STATE.G_Heating_Subsystem_Degraded OR GVL_STATE.G_DHW_Subsystem_Degraded OR GVL_STATE.G_Ventilation_Subsystem_Degraded OR GVL_STATUS.G_Diagnostics.Manifold_Pressure_Fault_Active OR GVL_STATUS.G_Diagnostics.Manifold_Current_Fault_Active OR GVL_STATUS.G_Diagnostics.Manifold_Return_Temp_Fault_Active
);

fbStateManager(
    VI_System_Severity := fbSystemHealth.VO_System_Severity,
    VI_Root_Cause := fbSystemHealth.VO_Root_Cause,
    VI_Freeze_Risk := GVL_STATE.G_Safety_Freeze_Risk
);

fbHMIInterface(
    VI_Severity := fbSystemHealth.VO_System_Severity,
    VI_RootCause := fbSystemHealth.VO_Root_Cause,
    VI_Status_Msg := fbStateManager.VO_Status_Msg
);

fbFaultLogger(
    VI_Severity := fbSystemHealth.VO_System_Severity,
    VI_RootCause := fbSystemHealth.VO_Root_Cause,
    VI_Time_MS := GVL_STATUS.G_System_Time_MS
);

GVL_STATUS.G_System_Mode_Msg := fbStateManager.VO_Status_Msg;

GVL_STATUS.G_Diagnostics.Sensor_Fault :=
    GVL_STATE.G_Heating_Sensor_Fault OR
    GVL_STATE.G_DHW_Sensor_Fault OR
    GVL_STATUS.G_Diagnostics.Manifold_Pressure_Fault_Active OR
    GVL_STATUS.G_Diagnostics.Manifold_Current_Fault_Active OR
    GVL_STATUS.G_Diagnostics.Manifold_Return_Temp_Fault_Active;

GVL_STATUS.G_Diagnostics.IO_Offline :=
    GVL_STATE.G_Heating_IO_Fault OR
    GVL_STATE.G_DHW_IO_Fault OR
    GVL_STATE.G_Ventilation_IO_Fault OR
    GVL_STATE.G_Lighting_IO_Fault;

GVL_STATUS.G_Diagnostics.Subsystem_Degraded :=
    GVL_STATE.G_Heating_Subsystem_Degraded OR
    GVL_STATE.G_DHW_Subsystem_Degraded OR
    GVL_STATE.G_Ventilation_Subsystem_Degraded OR
    GVL_STATUS.G_Diagnostics.Manifold_Pressure_Fault_Active OR
    GVL_STATUS.G_Diagnostics.Manifold_Current_Fault_Active OR
    GVL_STATUS.G_Diagnostics.Manifold_Return_Temp_Fault_Active;

GVL_GATEWAY.G_Gateway_HMI_Status_Message := fbHMIInterface.VO_HMI_Status_Text;
IF fbFaultLogger.VO_Last_Event_Text <> '' THEN
    GVL_HEALTH_BRIDGE.G_Last_Fault_Event_Text := fbFaultLogger.VO_Last_Event_Text;
END_IF;

GVL_STATE.G_System_Mode := fbStateManager.VO_System_Mode;

CASE GVL_STATE.G_System_Mode OF
    E_System_Operating_Mode.MODE_SAFE_STOP:
        GVL_STATE.G_System_Mode_Text := 'SAFE_STOP';

    E_System_Operating_Mode.MODE_FREEZE_PROTECTION:
        GVL_STATE.G_System_Mode_Text := 'FREEZE_PROTECTION';

    E_System_Operating_Mode.MODE_DEGRADED:
        GVL_STATE.G_System_Mode_Text := 'DEGRADED';

    ELSE
        GVL_STATE.G_System_Mode_Text := 'NORMAL';
END_CASE;

CASE fbSystemHealth.VO_Root_Cause OF
    E_System_Root_Cause.ROOT_FIRE:
        GVL_STATUS.G_System_Mode_Cause := 'Пожар/дым';
    E_System_Root_Cause.ROOT_GAS_LEAK:
        GVL_STATUS.G_System_Mode_Cause := 'Утечка газа';
    E_System_Root_Cause.ROOT_CO_CRITICAL:
        GVL_STATUS.G_System_Mode_Cause := 'Критический CO';
    E_System_Root_Cause.ROOT_CO_WARNING:
        GVL_STATUS.G_System_Mode_Cause := 'Повышенный CO';
    E_System_Root_Cause.ROOT_WATER_LEAK:
        GVL_STATUS.G_System_Mode_Cause := 'Протечка воды';
    E_System_Root_Cause.ROOT_WATCHDOG_FAULT:
        GVL_STATUS.G_System_Mode_Cause := 'Ошибка watchdog';
    E_System_Root_Cause.ROOT_IO_OFFLINE:
        GVL_STATUS.G_System_Mode_Cause := 'Недоступен модуль IO';
    E_System_Root_Cause.ROOT_COMM_FAULT:
        GVL_STATUS.G_System_Mode_Cause := 'Ошибка связи';
    E_System_Root_Cause.ROOT_SENSOR_FAULT:
        GVL_STATUS.G_System_Mode_Cause := 'Ошибка датчика';
    E_System_Root_Cause.ROOT_SUBSYSTEM_FAULT:
        GVL_STATUS.G_System_Mode_Cause := 'Ошибка подсистемы';
    ELSE
        GVL_STATUS.G_System_Mode_Cause := 'Аварийные режимы отсутствуют';
END_CASE;

VO_First_Fault_Active := fbSystemHealth.VO_First_Fault_Active;
VO_First_Fault_Type := fbSystemHealth.VO_First_Fault_Type;
VO_First_Fault_Source := fbSystemHealth.VO_First_Fault_Source;
VO_System_Severity := fbSystemHealth.VO_System_Severity;
VO_Root_Cause := fbSystemHealth.VO_Root_Cause;
VO_Watchdog_Fault := fbWatchdog.VO_Watchdog_Fault;

GVL_STATUS.G_System_Mode_Msg := fbStateManager.VO_Status_Msg;

// >>> BULK_SYNC_ANCHOR: FB_System_Health_Orchestrator <<<

(* ---- FB_System_History_Manager.st ---- *)
// ==============================================================================
// System history manager helper
//
// Internal helper for PRG_System.
// Owns history event detection, buffering, write index management,
// and interaction with FB_History_Manager.
// ==============================================================================
FUNCTION_BLOCK FB_System_History_Manager
VAR_INPUT
    VI_System_Time_MS : UDINT;
    VI_IsActivePLC : BOOL;
    VI_First_Fault_Active : BOOL;
    VI_First_Fault_Type : INT;
    VI_First_Fault_Source : INT;
END_VAR

VAR_IN_OUT
    VIO_History_Write_Event : BOOL;
    VIO_History_Write_Idx : INT;
    VIO_History_Total_Events : DINT;
    VIO_History_Buffer : ARRAY[0..255] OF ST_History_Event;
END_VAR

VAR
    fbHistoryManager : FB_History_Manager;
END_VAR

// Detect new history event
IF VI_First_Fault_Active THEN
    VIO_History_Write_Event := TRUE;
ELSE
    VIO_History_Write_Event := FALSE;
END_IF;

// Write event into buffer
IF VIO_History_Write_Event THEN
    VIO_History_Buffer[VIO_History_Write_Idx].Timestamp := VI_System_Time_MS;
    VIO_History_Buffer[VIO_History_Write_Idx].Fault_Type := VI_First_Fault_Type;
    VIO_History_Buffer[VIO_History_Write_Idx].Fault_Source := VI_First_Fault_Source;

    VIO_History_Write_Idx := VIO_History_Write_Idx + 1;
    IF VIO_History_Write_Idx > 255 THEN
        VIO_History_Write_Idx := 0;
    END_IF;

    VIO_History_Total_Events := VIO_History_Total_Events + 1;
END_IF;

// Call history manager
fbHistoryManager(
    VI_System_Time_MS := VI_System_Time_MS,
    VI_IsActivePLC := VI_IsActivePLC,
    VI_Write_Event := VIO_History_Write_Event,
    VIO_Write_Idx := VIO_History_Write_Idx,
    VIO_Total_Events := VIO_History_Total_Events,
    VIO_History_Buffer := VIO_History_Buffer
);

// >>> BULK_SYNC_ANCHOR: FB_System_History_Manager <<<

(* ---- FB_System_Init.st ---- *)
// ==============================================================================
// System init helper
//
// Internal helper for PRG_System.
// Owns first-boot initialization of RETAIN runtime state.
// ==============================================================================
FUNCTION_BLOCK FB_System_Init
VAR
    L_i : INT;
END_VAR

IF NOT GVL_Retain.G_Initialized THEN
    FOR L_i := 0 TO GVL_CONSTANTS.C_MAX_PRESENCE_HISTORY - 1 DO
        GVL_Retain.G_Presence_History[L_i] := 0;
    END_FOR;

    GVL_Retain.G_History_Write_Idx := 1;
    GVL_Retain.G_History_Total_Events := 0;

    FOR L_i := 1 TO GVL_CONSTANTS.C_MAX_BOILERS DO
        GVL_Retain.G_Boiler_Accumulated_MS[L_i] := 0;
        GVL_Retain.G_Boiler_Work_Seconds[L_i] := 0;
    END_FOR;

    FOR L_i := 1 TO GVL_CONSTANTS.C_MAX_MANIFOLDS DO
        GVL_Retain.G_Valve_Test_Results[L_i] := FALSE;
    END_FOR;

    GVL_Retain.G_Initialized := TRUE;
END_IF;

// >>> BULK_SYNC_ANCHOR: FB_System_Init <<<

(* ---- FB_System_Intent_Publisher.st ---- *)
// ==============================================================================
// System intent publisher helper
//
// Internal helper for PRG_System.
// Owns publication of system-mode gates into GVL_INTENT_SYSTEM.
// ==============================================================================
FUNCTION_BLOCK FB_System_Intent_Publisher
VAR_INPUT
    VI_System_Time_MS : UDINT;
    VI_Gateway_Writes_Allowed : BOOL;
END_VAR

GVL_INTENT_SYSTEM.I_Source_Valid := TRUE;
GVL_INTENT_SYSTEM.I_Last_Update_MS := VI_System_Time_MS;
GVL_INTENT_SYSTEM.I_Mode_Safe_Stop_Active := (GVL_STATE.G_System_Mode = E_System_Operating_Mode.MODE_SAFE_STOP);
GVL_INTENT_SYSTEM.I_Mode_Degraded_Active := (GVL_STATE.G_System_Mode = E_System_Operating_Mode.MODE_DEGRADED);
GVL_INTENT_SYSTEM.I_Mode_Freeze_Protection_Active := (GVL_STATE.G_System_Mode = E_System_Operating_Mode.MODE_FREEZE_PROTECTION);
GVL_INTENT_SYSTEM.I_Operator_Scenario_Block := (GVL_STATE.G_System_Mode = E_System_Operating_Mode.MODE_SAFE_STOP);
GVL_INTENT_SYSTEM.I_Lighting_Overrides_Block := (GVL_STATE.G_System_Mode = E_System_Operating_Mode.MODE_SAFE_STOP);
GVL_INTENT_SYSTEM.I_Blinds_Overrides_Block := (GVL_STATE.G_System_Mode = E_System_Operating_Mode.MODE_SAFE_STOP);
GVL_INTENT_SYSTEM.I_Socket_Overrides_Block := (GVL_STATE.G_System_Mode = E_System_Operating_Mode.MODE_SAFE_STOP);
GVL_INTENT_SYSTEM.I_Gateway_Writes_Allowed := VI_Gateway_Writes_Allowed;
GVL_INTENT_SYSTEM.I_Scenario_Request_Allowed := (GVL_STATE.G_System_Mode <> E_System_Operating_Mode.MODE_SAFE_STOP);

// >>> BULK_SYNC_ANCHOR: FB_System_Intent_Publisher <<<

(* ---- FB_System_Recovery.st ---- *)
// ==============================================================================
// System recovery helper
//
// Internal helper for PRG_System.
// Recovery no longer restores authoritative runtime state directly.
// Safety latches and system mode are reconstructed from current
// runtime truth through orchestrators/managers after boot.
// ==============================================================================
FUNCTION_BLOCK FB_System_Recovery
VAR_IN_OUT
    VIO_Recovery_Done : BOOL;
END_VAR

IF NOT VIO_Recovery_Done THEN
    VIO_Recovery_Done := TRUE;
END_IF;

// >>> BULK_SYNC_ANCHOR: FB_System_Recovery <<<
END_FUNCTION_BLOCK
